SPLINE
SPL {X  -159.990, Y  +513.606, Z    +0.000, E1  +339.879, E3 -411702.660}
SPL {X  -159.990, Y  +508.660, Z    +0.000, E1  +338.515, E3 -411718.090}
SPL {X  -159.990, Y  +505.237, Z    +0.000, E1  +337.606, E3 -411728.347}
SPL {X  -159.990, Y  +501.963, Z    +0.000, E1  +336.712, E3 -411737.451}
SPL {X  -159.990, Y  +498.406, Z    +0.000, E1  +335.789, E3 -411747.202}
SPL {X  -159.990, Y  +494.693, Z    +0.000, E1  +334.929, E3 -411757.669}
SPL {X  -159.990, Y  +491.649, Z    +0.000, E1  +334.596, E3 -411768.871}
SPL {X  -159.990, Y  +488.807, Z    +0.000, E1  +334.603, E3 -411781.596}
SPL {X  -159.990, Y  +486.070, Z    +0.000, E1  +334.601, E3 -411793.827}
SPL {X  -159.990, Y  +483.747, Z    +0.000, E1  +334.616, E3 -411804.240}
SPL {X  -159.990, Y  +481.980, Z    +0.000, E1  +334.616, E3 -411812.137}
SPL {X  -159.990, Y  +479.252, Z    +0.000, E1  +334.588, E3 -411824.279}
SPL {X  -159.990, Y  +475.940, Z    +0.000, E1  +334.597, E3 -411839.099}
SPL {X  -159.990, Y  +473.026, Z    +0.000, E1  +334.601, E3 -411852.129}
SPL {X  -159.990, Y  +470.047, Z    +0.000, E1  +334.598, E3 -411865.447}
SPL {X  -159.990, Y  +466.213, Z    +0.000, E1  +334.567, E3 -411882.527}
SPL {X  -159.990, Y  +462.520, Z    +0.000, E1  +334.600, E3 -411899.096}
SPL {X  -159.990, Y  +460.081, Z    +0.000, E1  +334.610, E3 -411909.997}
SPL {X  -159.990, Y  +457.497, Z    +0.000, E1  +334.597, E3 -411921.522}
SPL {X  -159.990, Y  +455.126, Z    +0.000, E1  +334.611, E3 -411932.130}
SPL {X  -159.990, Y  +452.123, Z    +0.000, E1  +334.574, E3 -411945.488}
SPL {X  -159.990, Y  +448.503, Z    +0.000, E1  +334.590, E3 -411961.689}
SPL {X  -159.990, Y  +445.882, Z    +0.000, E1  +334.615, E3 -411973.492}
SPL {X  -159.990, Y  +443.345, Z    +0.000, E1  +334.610, E3 -411984.874}
SPL {X  -159.990, Y  +441.077, Z    +0.000, E1  +334.631, E3 -411995.072}
SPL {X  -159.990, Y  +438.608, Z    +0.000, E1  +334.608, E3 -412006.069}
SPL {X  -159.990, Y  +435.579, Z    +0.000, E1  +334.614, E3 -412019.623}
SPL {X  -159.990, Y  +432.613, Z    +0.000, E1  +334.610, E3 -412032.890}
SPL {X  -159.990, Y  +429.079, Z    +0.000, E1  +334.593, E3 -412048.661}
SPL {X  -159.990, Y  +426.149, Z    +0.000, E1  +334.626, E3 -412061.823}
SPL {X  -159.990, Y  +423.417, Z    +0.000, E1  +334.600, E3 -412073.989}
SPL {X  -159.990, Y  +419.467, Z    +0.000, E1  +334.583, E3 -412091.623}
SPL {X  -159.990, Y  +416.355, Z    +0.000, E1  +334.625, E3 -412105.621}
SPL {X  -159.990, Y  +413.684, Z    +0.000, E1  +334.603, E3 -412117.527}
SPL {X  -159.990, Y  +410.645, Z    +0.000, E1  +334.615, E3 -412131.139}
SPL {X  -159.990, Y  +408.351, Z    +0.000, E1  +334.628, E3 -412141.425}
SPL {X  -159.990, Y  +406.574, Z    +0.000, E1  +334.625, E3 -412149.342}
SPL {X  -159.990, Y  +404.255, Z    +0.000, E1  +334.609, E3 -412159.678}
SPL {X  -159.990, Y  +401.103, Z    +0.000, E1  +334.596, E3 -412173.742}
SPL {X  -159.990, Y  +398.389, Z    +0.000, E1  +334.619, E3 -412185.938}
SPL {X  -159.990, Y  +395.411, Z    +0.000, E1  +334.600, E3 -412199.235}
SPL {X  -159.990, Y  +392.473, Z    +0.000, E1  +334.623, E3 -412212.421}
SPL {X  -159.990, Y  +390.187, Z    +0.000, E1  +334.622, E3 -412222.679}
SPL {X  -159.990, Y  +387.503, Z    +0.000, E1  +334.622, E3 -412234.673}
SPL {X  -159.990, Y  +384.711, Z    +0.000, E1  +334.612, E3 -412247.117}
SPL {X  -159.988, Y  +381.794, Z    +0.000, E1  +334.611, E3 -412260.152}
SPL {X  -159.958, Y  +379.279, Z    +0.000, E1  +334.625, E3 -412271.442}
SPL {X  -159.867, Y  +376.223, Z    +0.000, E1  +334.608, E3 -412285.157}
SPL {X  -159.727, Y  +373.325, Z    +0.000, E1  +334.659, E3 -412298.322}
SPL {X  -159.549, Y  +370.634, Z    +0.000, E1  +334.653, E3 -412310.495}
SPL {X  -159.201, Y  +366.633, Z    +0.000, E1  +334.686, E3 -412328.687}
SPL {X  -158.798, Y  +363.007, Z    +0.000, E1  +334.761, E3 -412345.345}
SPL {X  -158.453, Y  +360.380, Z    +0.000, E1  +334.828, E3 -412357.489}
SPL {X  -158.127, Y  +358.155, Z    +0.000, E1  +334.874, E3 -412367.820}
SPL {X  -158.095, Y  +357.947, Z    +0.000, E1  +338.259, E3 -412399.392}
ENDSPLINE

SPLINE
SPL {X  -158.454, Y  +360.384, Z    +0.000, E1  +340.634, E3 -412411.543}
SPL {X  -159.737, Y  +373.507, Z    +0.000, E1  +349.689, E3 -412433.579}
SPL {X  -159.990, Y  +382.574, Z    +0.000, E1  +355.537, E3 -412440.266}
SPL {X  -159.990, Y  +387.496, Z    +0.000, E1  +358.996, E3 -412443.012}
SPL {X  -159.990, Y  +395.121, Z    +0.000, E1  +364.514, E3 -412447.324}
SPL {X  -159.990, Y  +407.941, Z    +0.000, E1  +374.126, E3 -412459.398}
SPL {X  -159.990, Y  +418.671, Z    +0.000, E1  +379.855, E3 -412478.814}
SPL {X  -159.990, Y  +429.878, Z    +0.000, E1  +383.330, E3 -412508.869}
SPL {X  -159.990, Y  +432.766, Z    +0.000, E1  +383.321, E3 -412523.092}
SPL {X  -159.990, Y  +434.794, Z    +0.000, E1  +383.304, E3 -412533.123}
SPL {X  -159.990, Y  +437.007, Z    +0.000, E1  +383.323, E3 -412543.976}
SPL {X  -159.990, Y  +439.778, Z    +0.000, E1  +383.323, E3 -412557.608}
SPL {X  -159.990, Y  +442.010, Z    +0.000, E1  +383.308, E3 -412568.629}
SPL {X  -159.990, Y  +443.729, Z    +0.000, E1  +383.310, E3 -412577.085}
SPL {X  -159.990, Y  +446.037, Z    +0.000, E1  +383.324, E3 -412588.422}
SPL {X  -159.990, Y  +448.341, Z    +0.000, E1  +383.317, E3 -412599.740}
SPL {X  -159.990, Y  +450.345, Z    +0.000, E1  +383.316, E3 -412609.618}
SPL {X  -159.990, Y  +452.828, Z    +0.000, E1  +383.330, E3 -412621.817}
SPL {X  -159.990, Y  +456.338, Z    +0.000, E1  +383.359, E3 -412639.009}
SPL {X  -159.990, Y  +459.480, Z    +0.000, E1  +383.323, E3 -412654.551}
SPL {X  -159.990, Y  +461.803, Z    +0.000, E1  +383.322, E3 -412665.986}
SPL {X  -159.990, Y  +464.971, Z    +0.000, E1  +383.357, E3 -412681.492}
SPL {X  -159.990, Y  +467.934, Z    +0.000, E1  +383.321, E3 -412696.149}
SPL {X  -159.990, Y  +469.939, Z    +0.000, E1  +383.319, E3 -412706.011}
SPL {X  -159.990, Y  +472.144, Z    +0.000, E1  +383.327, E3 -412716.862}
SPL {X  -159.990, Y  +474.152, Z    +0.000, E1  +383.309, E3 -412726.814}
SPL {X  -159.990, Y  +476.560, Z    +0.000, E1  +383.332, E3 -412738.622}
SPL {X  -159.990, Y  +478.770, Z    +0.000, E1  +383.306, E3 -412749.547}
SPL {X  -159.990, Y  +480.905, Z    +0.000, E1  +383.327, E3 -412760.015}
SPL {X  -159.990, Y  +484.251, Z    +0.000, E1  +383.352, E3 -412776.430}
SPL {X  -159.990, Y  +488.031, Z    +0.000, E1  +383.345, E3 -412795.063}
SPL {X  -159.990, Y  +491.121, Z    +0.000, E1  +383.323, E3 -412810.309}
SPL {X  -159.990, Y  +493.610, Z    +0.000, E1  +383.323, E3 -412822.562}
SPL {X  -159.990, Y  +496.863, Z    +0.000, E1  +383.350, E3 -412838.522}
SPL {X  -159.990, Y  +499.995, Z    +0.000, E1  +383.324, E3 -412853.983}
SPL {X  -159.990, Y  +502.341, Z    +0.000, E1  +383.320, E3 -412865.542}
SPL {X  -159.990, Y  +504.419, Z    +0.000, E1  +383.313, E3 -412875.784}
SPL {X  -159.990, Y  +507.187, Z    +0.000, E1  +383.346, E3 -412889.337}
SPL {X  -159.990, Y  +510.344, Z    +0.000, E1  +383.327, E3 -412904.922}
SPL {X  -159.990, Y  +512.484, Z    +0.000, E1  +383.309, E3 -412915.494}
SPL {X  -159.990, Y  +514.016, Z    +0.000, E1  +383.308, E3 -412923.043}
SPL {X  -159.990, Y  +516.195, Z    +0.000, E1  +383.325, E3 -412933.731}
SPL {X  -159.990, Y  +518.925, Z    +0.000, E1  +383.333, E3 -412947.094}
SPL {X  -159.990, Y  +521.408, Z    +0.000, E1  +383.329, E3 -412959.303}
SPL {X  -159.990, Y  +523.942, Z    +0.000, E1  +383.333, E3 -412971.796}
SPL {X  -159.990, Y  +527.007, Z    +0.000, E1  +383.339, E3 -412986.895}
SPL {X  -159.990, Y  +529.993, Z    +0.000, E1  +383.329, E3 -413001.598}
SPL {X  -159.990, Y  +532.441, Z    +0.000, E1  +383.322, E3 -413013.649}
SPL {X  -159.990, Y  +534.618, Z    +0.000, E1  +383.322, E3 -413024.382}
SPL {X  -159.990, Y  +537.024, Z    +0.000, E1  +383.321, E3 -413036.244}
SPL {X  -159.990, Y  +539.129, Z    +0.000, E1  +383.310, E3 -413046.627}
SPL {X  -159.990, Y  +541.183, Z    +0.000, E1  +383.319, E3 -413056.724}
SPL {X  -159.990, Y  +543.647, Z    +0.000, E1  +383.325, E3 -413068.827}
SPL {X  -159.990, Y  +546.832, Z    +0.000, E1  +383.349, E3 -413084.450}
SPL {X  -159.990, Y  +549.756, Z    +0.000, E1  +383.320, E3 -413098.891}
SPL {X  -159.990, Y  +551.655, Z    +0.000, E1  +383.320, E3 -413108.241}
SPL {X  -159.990, Y  +553.711, Z    +0.000, E1  +383.317, E3 -413118.363}
SPL {X  -159.990, Y  +556.481, Z    +0.000, E1  +383.354, E3 -413131.925}
SPL {X  -159.990, Y  +559.475, Z    +0.000, E1  +383.321, E3 -413146.730}
SPL {X  -159.990, Y  +561.830, Z    +0.000, E1  +383.325, E3 -413158.315}
SPL {X  -159.990, Y  +564.273, Z    +0.000, E1  +383.325, E3 -413170.339}
SPL {X  -159.990, Y  +566.342, Z    +0.000, E1  +383.314, E3 -413180.544}
SPL {X  -159.990, Y  +568.184, Z    +0.000, E1  +383.317, E3 -413189.605}
SPL {X  -159.990, Y  +570.314, Z    +0.000, E1  +383.326, E3 -413200.067}
SPL {X  -159.990, Y  +573.444, Z    +0.000, E1  +383.356, E3 -413215.406}
SPL {X  -159.990, Y  +577.161, Z    +0.000, E1  +383.346, E3 -413233.731}
SPL {X  -159.990, Y  +580.840, Z    +0.000, E1  +383.355, E3 -413251.780}
SPL {X  -159.990, Y  +583.973, Z    +0.000, E1  +383.332, E3 -413267.241}
SPL {X  -159.990, Y  +586.020, Z    +0.000, E1  +383.323, E3 -413277.325}
SPL {X  -159.990, Y  +587.711, Z    +0.000, E1  +383.318, E3 -413285.665}
SPL {X  -159.990, Y  +589.763, Z    +0.000, E1  +383.328, E3 -413295.741}
SPL {X  -159.990, Y  +591.698, Z    +0.000, E1  +383.324, E3 -413305.226}
SPL {X  -159.990, Y  +593.847, Z    +0.000, E1  +383.340, E3 -413315.757}
SPL {X  -159.990, Y  +597.018, Z    +0.000, E1  +383.367, E3 -413331.288}
SPL {X  -159.990, Y  +599.887, Z    +0.000, E1  +383.341, E3 -413345.393}
SPL {X  -159.990, Y  +601.949, Z    +0.000, E1  +383.344, E3 -413355.519}
SPL {X  -159.990, Y  +605.106, Z    +0.000, E1  +383.383, E3 -413370.965}
SPL {X  -159.990, Y  +608.111, Z    +0.000, E1  +383.342, E3 -413385.816}
SPL {X  -159.990, Y  +610.073, Z    +0.000, E1  +383.343, E3 -413395.474}
SPL {X  -159.990, Y  +612.330, Z    +0.000, E1  +383.340, E3 -413406.602}
SPL {X  -159.990, Y  +615.036, Z    +0.000, E1  +383.353, E3 -413419.889}
SPL {X  -159.990, Y  +618.481, Z    +0.000, E1  +383.366, E3 -413436.827}
SPL {X  -159.990, Y  +621.517, Z    +0.000, E1  +383.337, E3 -413451.810}
SPL {X  -159.990, Y  +623.764, Z    +0.000, E1  +383.335, E3 -413462.861}
SPL {X  -159.990, Y  +626.608, Z    +0.000, E1  +383.361, E3 -413476.786}
SPL {X  -159.990, Y  +630.271, Z    +0.000, E1  +383.375, E3 -413494.747}
SPL {X  -159.990, Y  +633.318, Z    +0.000, E1  +383.339, E3 -413509.824}
SPL {X  -159.990, Y  +635.650, Z    +0.000, E1  +383.339, E3 -413521.295}
SPL {X  -159.990, Y  +638.406, Z    +0.000, E1  +383.354, E3 -413534.862}
SPL {X  -159.990, Y  +641.831, Z    +0.000, E1  +383.342, E3 -413551.809}
SPL {X  -159.990, Y  +644.884, Z    +0.000, E1  +383.324, E3 -413566.896}
SPL {X  -159.990, Y  +647.550, Z    +0.000, E1  +383.318, E3 -413580.063}
SPL {X  -159.990, Y  +650.790, Z    +0.000, E1  +383.346, E3 -413595.930}
SPL {X  -159.990, Y  +654.543, Z    +0.000, E1  +383.348, E3 -413614.382}
SPL {X  -159.990, Y  +658.319, Z    +0.000, E1  +383.349, E3 -413632.972}
SPL {X  -159.990, Y  +661.392, Z    +0.000, E1  +383.318, E3 -413648.175}
SPL {X  -159.990, Y  +663.662, Z    +0.000, E1  +383.322, E3 -413659.299}
SPL {X  -159.990, Y  +665.964, Z    +0.000, E1  +383.328, E3 -413670.590}
SPL {X  -159.990, Y  +667.870, Z    +0.000, E1  +383.320, E3 -413679.996}
SPL {X  -159.990, Y  +669.861, Z    +0.000, E1  +383.321, E3 -413689.798}
SPL {X  -159.983, Y  +672.946, Z    +0.000, E1  +383.359, E3 -413704.907}
SPL {X  -159.924, Y  +676.110, Z    +0.000, E1  +383.320, E3 -413720.606}
SPL {X  -159.845, Y  +678.302, Z    +0.000, E1  +383.298, E3 -413731.508}
SPL {X  -159.760, Y  +680.081, Z    +0.000, E1  +383.288, E3 -413740.352}
SPL {X  -159.626, Y  +682.287, Z    +0.000, E1  +383.280, E3 -413751.323}
SPL {X  -159.462, Y  +684.486, Z    +0.000, E1  +383.258, E3 -413762.323}
SPL {X  -159.212, Y  +687.262, Z    +0.000, E1  +383.238, E3 -413776.227}
SPL {X  -158.971, Y  +689.529, Z    +0.000, E1  +383.181, E3 -413787.686}
SPL {X  -158.658, Y  +692.098, Z    +0.000, E1  +383.176, E3 -413800.593}
ENDSPLINE

SPLINE
SPL {X  -159.063, Y  +688.696, Z    +0.000, E1  +377.094, E3 -413842.811}
SPL {X  -159.987, Y  +672.488, Z    +0.000, E1  +365.638, E3 -413866.876}
SPL {X  -159.990, Y  +663.928, Z    +0.000, E1  +359.662, E3 -413872.671}
SPL {X  -159.990, Y  +658.009, Z    +0.000, E1  +355.226, E3 -413876.371}
SPL {X  -159.990, Y  +651.879, Z    +0.000, E1  +350.548, E3 -413881.433}
SPL {X  -159.990, Y  +637.832, Z    +0.000, E1  +341.694, E3 -413899.024}
SPL {X  -159.990, Y  +626.634, Z    +0.000, E1  +337.968, E3 -413929.877}
SPL {X  -159.990, Y  +624.622, Z    +0.000, E1  +337.980, E3 -413940.461}
SPL {X  -159.990, Y  +622.489, Z    +0.000, E1  +337.969, E3 -413951.628}
SPL {X  -159.990, Y  +619.955, Z    +0.000, E1  +337.968, E3 -413964.918}
SPL {X  -159.990, Y  +617.386, Z    +0.000, E1  +337.968, E3 -413978.392}
SPL {X  -159.990, Y  +614.863, Z    +0.000, E1  +337.969, E3 -413991.625}
SPL {X  -159.990, Y  +612.600, Z    +0.000, E1  +337.975, E3 -414003.509}
SPL {X  -159.990, Y  +610.646, Z    +0.000, E1  +337.979, E3 -414013.766}
SPL {X  -159.990, Y  +608.810, Z    +0.000, E1  +337.977, E3 -414023.399}
SPL {X  -159.990, Y  +605.804, Z    +0.000, E1  +337.936, E3 -414039.044}
SPL {X  -159.990, Y  +602.819, Z    +0.000, E1  +337.963, E3 -414054.715}
SPL {X  -159.990, Y  +600.642, Z    +0.000, E1  +337.968, E3 -414066.143}
SPL {X  -159.990, Y  +598.568, Z    +0.000, E1  +337.954, E3 -414076.936}
SPL {X  -159.990, Y  +596.440, Z    +0.000, E1  +337.964, E3 -414088.118}
SPL {X  -159.990, Y  +593.768, Z    +0.000, E1  +337.929, E3 -414102.051}
SPL {X  -159.990, Y  +590.068, Z    +0.000, E1  +337.924, E3 -414121.419}
SPL {X  -159.990, Y  +586.620, Z    +0.000, E1  +337.935, E3 -414139.482}
SPL {X  -159.990, Y  +584.080, Z    +0.000, E1  +337.953, E3 -414152.808}
SPL {X  -159.990, Y  +581.924, Z    +0.000, E1  +337.949, E3 -414164.108}
SPL {X  -159.990, Y  +578.886, Z    +0.000, E1  +337.918, E3 -414179.962}
SPL {X  -159.990, Y  +576.252, Z    +0.000, E1  +337.962, E3 -414193.860}
SPL {X  -159.990, Y  +574.188, Z    +0.000, E1  +337.947, E3 -414204.633}
SPL {X  -159.990, Y  +571.954, Z    +0.000, E1  +337.959, E3 -414216.391}
SPL {X  -159.990, Y  +570.110, Z    +0.000, E1  +337.958, E3 -414226.041}
SPL {X  -159.990, Y  +568.165, Z    +0.000, E1  +337.957, E3 -414236.221}
SPL {X  -159.990, Y  +566.106, Z    +0.000, E1  +337.954, E3 -414247.004}
SPL {X  -159.990, Y  +563.259, Z    +0.000, E1  +337.929, E3 -414261.886}
SPL {X  -159.990, Y  +559.661, Z    +0.000, E1  +337.922, E3 -414280.709}
SPL {X  -159.990, Y  +555.965, Z    +0.000, E1  +337.915, E3 -414300.018}
SPL {X  -159.990, Y  +553.115, Z    +0.000, E1  +337.946, E3 -414315.003}
SPL {X  -159.990, Y  +550.886, Z    +0.000, E1  +337.944, E3 -414326.685}
SPL {X  -159.990, Y  +548.568, Z    +0.000, E1  +337.944, E3 -414338.806}
SPL {X  -159.990, Y  +545.859, Z    +0.000, E1  +337.926, E3 -414352.955}
SPL {X  -159.990, Y  +543.060, Z    +0.000, E1  +337.943, E3 -414367.679}
SPL {X  -159.990, Y  +539.928, Z    +0.000, E1  +337.917, E3 -414384.020}
SPL {X  -159.990, Y  +536.935, Z    +0.000, E1  +337.942, E3 -414399.737}
SPL {X  -159.990, Y  +534.656, Z    +0.000, E1  +337.946, E3 -414411.681}
SPL {X  -159.990, Y  +531.679, Z    +0.000, E1  +337.913, E3 -414427.195}
SPL {X  -159.990, Y  +527.941, Z    +0.000, E1  +337.907, E3 -414446.737}
SPL {X  -159.990, Y  +525.053, Z    +0.000, E1  +337.942, E3 -414461.927}
SPL {X  -159.990, Y  +522.838, Z    +0.000, E1  +337.933, E3 -414473.531}
SPL {X  -159.990, Y  +519.698, Z    +0.000, E1  +337.916, E3 -414489.915}
SPL {X  -159.990, Y  +517.251, Z    +0.000, E1  +337.946, E3 -414502.774}
SPL {X  -159.990, Y  +515.568, Z    +0.000, E1  +338.084, E3 -414512.871}
ENDSPLINE

SPLINE
SPL {X  -159.990, Y  +517.293, Z    +0.000, E1  +340.923, E3 -414529.170}
ENDSPLINE

SPLINE
SPL {X  -159.990, Y  +512.548, Z    +0.000, E1  +339.587, E3 -414544.745}
SPL {X  -159.990, Y  +508.660, Z    +0.000, E1  +338.515, E3 -414556.799}
SPL {X  -159.990, Y  +503.499, Z    +0.000, E1  +337.116, E3 -414571.878}
SPL {X  -159.990, Y  +498.406, Z    +0.000, E1  +335.789, E3 -414585.911}
SPL {X  -159.990, Y  +494.693, Z    +0.000, E1  +334.929, E3 -414596.379}
SPL {X  -159.990, Y  +491.649, Z    +0.000, E1  +334.596, E3 -414607.581}
SPL {X  -159.990, Y  +488.807, Z    +0.000, E1  +334.603, E3 -414620.306}
SPL {X  -159.990, Y  +486.070, Z    +0.000, E1  +334.601, E3 -414632.537}
SPL {X  -159.990, Y  +482.821, Z    +0.000, E1  +334.589, E3 -414647.038}
SPL {X  -159.990, Y  +480.183, Z    +0.000, E1  +334.616, E3 -414658.878}
SPL {X  -159.990, Y  +478.407, Z    +0.000, E1  +334.616, E3 -414666.819}
SPL {X  -159.990, Y  +475.940, Z    +0.000, E1  +334.597, E3 -414677.809}
SPL {X  -159.990, Y  +473.026, Z    +0.000, E1  +334.601, E3 -414690.839}
SPL {X  -159.990, Y  +470.047, Z    +0.000, E1  +334.598, E3 -414704.157}
SPL {X  -159.990, Y  +467.082, Z    +0.000, E1  +334.601, E3 -414717.404}
SPL {X  -159.990, Y  +464.919, Z    +0.000, E1  +334.619, E3 -414727.131}
SPL {X  -159.990, Y  +462.520, Z    +0.000, E1  +334.600, E3 -414737.805}
SPL {X  -159.990, Y  +460.081, Z    +0.000, E1  +334.610, E3 -414748.707}
SPL {X  -159.990, Y  +457.497, Z    +0.000, E1  +334.597, E3 -414760.231}
SPL {X  -159.990, Y  +454.323, Z    +0.000, E1  +334.588, E3 -414774.390}
SPL {X  -159.990, Y  +451.400, Z    +0.000, E1  +334.603, E3 -414787.481}
SPL {X  -159.990, Y  +448.503, Z    +0.000, E1  +334.590, E3 -414800.399}
SPL {X  -159.990, Y  +445.108, Z    +0.000, E1  +334.593, E3 -414815.637}
SPL {X  -159.990, Y  +441.797, Z    +0.000, E1  +334.610, E3 -414830.516}
SPL {X  -159.990, Y  +439.442, Z    +0.000, E1  +334.631, E3 -414841.093}
SPL {X  -159.990, Y  +436.316, Z    +0.000, E1  +334.580, E3 -414854.975}
SPL {X  -159.990, Y  +432.613, Z    +0.000, E1  +334.610, E3 -414871.600}
SPL {X  -159.990, Y  +429.079, Z    +0.000, E1  +334.593, E3 -414887.371}
SPL {X  -159.990, Y  +426.149, Z    +0.000, E1  +334.626, E3 -414900.533}
SPL {X  -159.990, Y  +423.417, Z    +0.000, E1  +334.600, E3 -414912.698}
SPL {X  -159.990, Y  +419.467, Z    +0.000, E1  +334.583, E3 -414930.333}
SPL {X  -159.990, Y  +416.355, Z    +0.000, E1  +334.625, E3 -414944.330}
SPL {X  -159.990, Y  +413.684, Z    +0.000, E1  +334.603, E3 -414956.237}
SPL {X  -159.990, Y  +410.645, Z    +0.000, E1  +334.615, E3 -414969.849}
SPL {X  -159.990, Y  +408.351, Z    +0.000, E1  +334.628, E3 -414980.135}
SPL {X  -159.990, Y  +406.574, Z    +0.000, E1  +334.625, E3 -414988.052}
SPL {X  -159.990, Y  +404.255, Z    +0.000, E1  +334.609, E3 -414998.388}
SPL {X  -159.990, Y  +401.103, Z    +0.000, E1  +334.596, E3 -415012.452}
SPL {X  -159.990, Y  +398.389, Z    +0.000, E1  +334.619, E3 -415024.648}
SPL {X  -159.990, Y  +395.411, Z    +0.000, E1  +334.600, E3 -415037.945}
SPL {X  -159.990, Y  +392.473, Z    +0.000, E1  +334.623, E3 -415051.130}
SPL {X  -159.990, Y  +390.187, Z    +0.000, E1  +334.622, E3 -415061.388}
SPL {X  -159.990, Y  +387.503, Z    +0.000, E1  +334.622, E3 -415073.383}
SPL {X  -159.990, Y  +384.711, Z    +0.000, E1  +334.612, E3 -415085.827}
SPL {X  -159.988, Y  +381.794, Z    +0.000, E1  +334.611, E3 -415098.862}
SPL {X  -159.958, Y  +379.279, Z    +0.000, E1  +334.625, E3 -415110.152}
SPL {X  -159.894, Y  +376.959, Z    +0.000, E1  +334.630, E3 -415120.596}
SPL {X  -159.765, Y  +374.027, Z    +0.000, E1  +334.633, E3 -415133.812}
SPL {X  -159.607, Y  +371.442, Z    +0.000, E1  +334.673, E3 -415145.587}
SPL {X  -159.379, Y  +368.534, Z    +0.000, E1  +334.684, E3 -415158.774}
SPL {X  -159.113, Y  +365.767, Z    +0.000, E1  +334.734, E3 -415171.414}
SPL {X  -158.869, Y  +363.595, Z    +0.000, E1  +334.770, E3 -415181.385}
SPL {X  -158.527, Y  +360.915, Z    +0.000, E1  +334.798, E3 -415193.692}
SPL {X  -158.127, Y  +358.155, Z    +0.000, E1  +334.874, E3 -415206.530}
SPL {X  -158.095, Y  +357.947, Z    +0.000, E1  +338.259, E3 -415238.102}
ENDSPLINE

SPLINE
SPL {X  -158.454, Y  +360.384, Z    +0.000, E1  +340.634, E3 -415250.253}
SPL {X  -159.737, Y  +373.507, Z    +0.000, E1  +349.689, E3 -415272.288}
SPL {X  -159.990, Y  +382.574, Z    +0.000, E1  +355.537, E3 -415278.976}
SPL {X  -159.990, Y  +387.496, Z    +0.000, E1  +358.996, E3 -415281.721}
SPL {X  -159.990, Y  +395.121, Z    +0.000, E1  +364.514, E3 -415286.033}
SPL {X  -159.990, Y  +407.941, Z    +0.000, E1  +374.126, E3 -415298.108}
SPL {X  -159.990, Y  +418.671, Z    +0.000, E1  +379.855, E3 -415317.524}
SPL {X  -159.990, Y  +429.878, Z    +0.000, E1  +383.330, E3 -415347.579}
SPL {X  -159.990, Y  +432.103, Z    +0.000, E1  +383.301, E3 -415358.598}
SPL {X  -159.990, Y  +434.188, Z    +0.000, E1  +383.325, E3 -415368.794}
SPL {X  -159.990, Y  +436.320, Z    +0.000, E1  +383.304, E3 -415379.347}
SPL {X  -159.990, Y  +439.169, Z    +0.000, E1  +383.353, E3 -415393.264}
SPL {X  -159.990, Y  +442.945, Z    +0.000, E1  +383.339, E3 -415411.882}
SPL {X  -159.990, Y  +446.037, Z    +0.000, E1  +383.324, E3 -415427.132}
SPL {X  -159.990, Y  +448.341, Z    +0.000, E1  +383.317, E3 -415438.449}
SPL {X  -159.990, Y  +450.345, Z    +0.000, E1  +383.316, E3 -415448.327}
SPL {X  -159.990, Y  +452.828, Z    +0.000, E1  +383.330, E3 -415460.527}
SPL {X  -159.990, Y  +456.338, Z    +0.000, E1  +383.359, E3 -415477.719}
SPL {X  -159.990, Y  +459.480, Z    +0.000, E1  +383.323, E3 -415493.260}
SPL {X  -159.990, Y  +461.803, Z    +0.000, E1  +383.322, E3 -415504.695}
SPL {X  -159.990, Y  +464.971, Z    +0.000, E1  +383.357, E3 -415520.201}
SPL {X  -159.990, Y  +467.934, Z    +0.000, E1  +383.321, E3 -415534.859}
SPL {X  -159.990, Y  +469.939, Z    +0.000, E1  +383.319, E3 -415544.720}
SPL {X  -159.990, Y  +472.144, Z    +0.000, E1  +383.327, E3 -415555.571}
SPL {X  -159.990, Y  +474.152, Z    +0.000, E1  +383.309, E3 -415565.523}
SPL {X  -159.990, Y  +475.762, Z    +0.000, E1  +383.308, E3 -415573.453}
SPL {X  -159.990, Y  +478.041, Z    +0.000, E1  +383.328, E3 -415584.628}
SPL {X  -159.990, Y  +480.905, Z    +0.000, E1  +383.327, E3 -415598.724}
SPL {X  -159.990, Y  +483.391, Z    +0.000, E1  +383.320, E3 -415610.965}
SPL {X  -159.990, Y  +485.299, Z    +0.000, E1  +383.310, E3 -415620.394}
SPL {X  -159.990, Y  +487.362, Z    +0.000, E1  +383.320, E3 -415630.528}
SPL {X  -159.990, Y  +490.503, Z    +0.000, E1  +383.351, E3 -415645.923}
SPL {X  -159.990, Y  +493.610, Z    +0.000, E1  +383.323, E3 -415661.272}
SPL {X  -159.990, Y  +495.794, Z    +0.000, E1  +383.312, E3 -415672.045}
SPL {X  -159.990, Y  +497.668, Z    +0.000, E1  +383.317, E3 -415681.255}
SPL {X  -159.990, Y  +499.995, Z    +0.000, E1  +383.324, E3 -415692.693}
SPL {X  -159.990, Y  +502.341, Z    +0.000, E1  +383.320, E3 -415704.252}
SPL {X  -159.990, Y  +504.419, Z    +0.000, E1  +383.313, E3 -415714.493}
SPL {X  -159.990, Y  +506.252, Z    +0.000, E1  +383.313, E3 -415723.519}
SPL {X  -159.990, Y  +508.697, Z    +0.000, E1  +383.335, E3 -415735.502}
SPL {X  -159.990, Y  +511.771, Z    +0.000, E1  +383.331, E3 -415750.649}
SPL {X  -159.990, Y  +514.016, Z    +0.000, E1  +383.308, E3 -415761.753}
SPL {X  -159.990, Y  +516.195, Z    +0.000, E1  +383.325, E3 -415772.440}
SPL {X  -159.990, Y  +518.925, Z    +0.000, E1  +383.333, E3 -415785.804}
SPL {X  -159.990, Y  +521.408, Z    +0.000, E1  +383.329, E3 -415798.013}
SPL {X  -159.990, Y  +523.942, Z    +0.000, E1  +383.333, E3 -415810.506}
SPL {X  -159.990, Y  +526.221, Z    +0.000, E1  +383.314, E3 -415821.782}
SPL {X  -159.990, Y  +527.834, Z    +0.000, E1  +383.311, E3 -415829.732}
SPL {X  -159.990, Y  +529.993, Z    +0.000, E1  +383.329, E3 -415840.308}
SPL {X  -159.990, Y  +532.441, Z    +0.000, E1  +383.322, E3 -415852.358}
SPL {X  -159.990, Y  +534.618, Z    +0.000, E1  +383.322, E3 -415863.091}
SPL {X  -159.990, Y  +537.024, Z    +0.000, E1  +383.321, E3 -415874.954}
SPL {X  -159.990, Y  +539.129, Z    +0.000, E1  +383.310, E3 -415885.337}
SPL {X  -159.990, Y  +541.183, Z    +0.000, E1  +383.319, E3 -415895.433}
SPL {X  -159.990, Y  +543.647, Z    +0.000, E1  +383.325, E3 -415907.536}
SPL {X  -159.990, Y  +546.832, Z    +0.000, E1  +383.349, E3 -415923.159}
SPL {X  -159.990, Y  +549.756, Z    +0.000, E1  +383.320, E3 -415937.600}
SPL {X  -159.990, Y  +551.655, Z    +0.000, E1  +383.320, E3 -415946.951}
SPL {X  -159.990, Y  +553.711, Z    +0.000, E1  +383.317, E3 -415957.073}
SPL {X  -159.990, Y  +555.637, Z    +0.000, E1  +383.323, E3 -415966.542}
SPL {X  -159.990, Y  +558.758, Z    +0.000, E1  +383.351, E3 -415981.851}
SPL {X  -159.990, Y  +561.830, Z    +0.000, E1  +383.325, E3 -415997.025}
SPL {X  -159.990, Y  +564.273, Z    +0.000, E1  +383.325, E3 -416009.049}
SPL {X  -159.990, Y  +567.351, Z    +0.000, E1  +383.348, E3 -416024.145}
SPL {X  -159.990, Y  +570.314, Z    +0.000, E1  +383.326, E3 -416038.777}
SPL {X  -159.990, Y  +572.504, Z    +0.000, E1  +383.321, E3 -416049.562}
SPL {X  -159.990, Y  +575.653, Z    +0.000, E1  +383.355, E3 -416064.999}
SPL {X  -159.990, Y  +578.932, Z    +0.000, E1  +383.330, E3 -416081.181}
SPL {X  -159.990, Y  +581.497, Z    +0.000, E1  +383.329, E3 -416093.766}
SPL {X  -159.990, Y  +583.973, Z    +0.000, E1  +383.332, E3 -416105.951}
SPL {X  -159.990, Y  +586.020, Z    +0.000, E1  +383.323, E3 -416116.035}
SPL {X  -159.990, Y  +587.711, Z    +0.000, E1  +383.318, E3 -416124.375}
SPL {X  -159.990, Y  +589.763, Z    +0.000, E1  +383.328, E3 -416134.451}
SPL {X  -159.990, Y  +591.698, Z    +0.000, E1  +383.324, E3 -416143.936}
SPL {X  -159.990, Y  +593.847, Z    +0.000, E1  +383.340, E3 -416154.466}
SPL {X  -159.990, Y  +597.018, Z    +0.000, E1  +383.367, E3 -416169.998}
SPL {X  -159.990, Y  +599.887, Z    +0.000, E1  +383.341, E3 -416184.102}
SPL {X  -159.990, Y  +601.949, Z    +0.000, E1  +383.344, E3 -416194.229}
SPL {X  -159.990, Y  +605.106, Z    +0.000, E1  +383.383, E3 -416209.675}
SPL {X  -159.990, Y  +608.111, Z    +0.000, E1  +383.342, E3 -416224.526}
SPL {X  -159.990, Y  +610.073, Z    +0.000, E1  +383.343, E3 -416234.184}
SPL {X  -159.990, Y  +612.330, Z    +0.000, E1  +383.340, E3 -416245.312}
SPL {X  -159.990, Y  +615.036, Z    +0.000, E1  +383.353, E3 -416258.599}
SPL {X  -159.990, Y  +618.481, Z    +0.000, E1  +383.366, E3 -416275.537}
SPL {X  -159.990, Y  +621.517, Z    +0.000, E1  +383.337, E3 -416290.520}
SPL {X  -159.990, Y  +623.764, Z    +0.000, E1  +383.335, E3 -416301.570}
SPL {X  -159.990, Y  +626.608, Z    +0.000, E1  +383.361, E3 -416315.495}
SPL {X  -159.990, Y  +630.271, Z    +0.000, E1  +383.375, E3 -416333.456}
SPL {X  -159.990, Y  +633.318, Z    +0.000, E1  +383.339, E3 -416348.534}
SPL {X  -159.990, Y  +635.650, Z    +0.000, E1  +383.339, E3 -416360.005}
SPL {X  -159.990, Y  +638.406, Z    +0.000, E1  +383.354, E3 -416373.571}
SPL {X  -159.990, Y  +641.131, Z    +0.000, E1  +383.320, E3 -416387.096}
SPL {X  -159.990, Y  +644.241, Z    +0.000, E1  +383.355, E3 -416402.374}
SPL {X  -159.990, Y  +648.287, Z    +0.000, E1  +383.349, E3 -416422.331}
SPL {X  -159.990, Y  +651.427, Z    +0.000, E1  +383.319, E3 -416437.826}
SPL {X  -159.990, Y  +653.536, Z    +0.000, E1  +383.313, E3 -416448.207}
SPL {X  -159.990, Y  +656.380, Z    +0.000, E1  +383.347, E3 -416462.143}
SPL {X  -159.990, Y  +659.180, Z    +0.000, E1  +383.314, E3 -416475.991}
SPL {X  -159.990, Y  +661.392, Z    +0.000, E1  +383.318, E3 -416486.885}
SPL {X  -159.990, Y  +663.662, Z    +0.000, E1  +383.322, E3 -416498.009}
SPL {X  -159.990, Y  +665.964, Z    +0.000, E1  +383.328, E3 -416509.299}
SPL {X  -159.990, Y  +668.989, Z    +0.000, E1  +383.359, E3 -416524.135}
SPL {X  -159.983, Y  +672.946, Z    +0.000, E1  +383.359, E3 -416543.616}
SPL {X  -159.924, Y  +676.110, Z    +0.000, E1  +383.320, E3 -416559.316}
SPL {X  -159.845, Y  +678.302, Z    +0.000, E1  +383.298, E3 -416570.218}
SPL {X  -159.760, Y  +680.081, Z    +0.000, E1  +383.288, E3 -416579.061}
SPL {X  -159.626, Y  +682.287, Z    +0.000, E1  +383.280, E3 -416590.033}
SPL {X  -159.462, Y  +684.486, Z    +0.000, E1  +383.258, E3 -416601.032}
SPL {X  -159.289, Y  +686.457, Z    +0.000, E1  +383.223, E3 -416610.943}
SPL {X  -159.052, Y  +688.801, Z    +0.000, E1  +383.217, E3 -416622.677}
SPL {X  -158.770, Y  +691.222, Z    +0.000, E1  +383.158, E3 -416634.935}
SPL {X  -158.553, Y  +692.896, Z    +0.000, E1  +383.130, E3 -416643.400}
ENDSPLINE

SPLINE
SPL {X  -158.898, Y  +690.164, Z    +0.000, E1  +378.236, E3 -416676.756}
SPL {X  -159.149, Y  +687.882, Z    +0.000, E1  +376.368, E3 -416684.044}
SPL {X  -159.987, Y  +672.488, Z    +0.000, E1  +365.638, E3 -416705.586}
SPL {X  -159.990, Y  +663.928, Z    +0.000, E1  +359.662, E3 -416711.381}
SPL {X  -159.990, Y  +658.009, Z    +0.000, E1  +355.226, E3 -416715.080}
SPL {X  -159.990, Y  +651.879, Z    +0.000, E1  +350.548, E3 -416720.143}
SPL {X  -159.990, Y  +637.832, Z    +0.000, E1  +341.694, E3 -416737.734}
SPL {X  -159.990, Y  +626.634, Z    +0.000, E1  +337.968, E3 -416768.587}
SPL {X  -159.990, Y  +624.622, Z    +0.000, E1  +337.980, E3 -416779.171}
SPL {X  -159.990, Y  +622.489, Z    +0.000, E1  +337.969, E3 -416790.337}
SPL {X  -159.990, Y  +619.955, Z    +0.000, E1  +337.968, E3 -416803.627}
SPL {X  -159.990, Y  +617.386, Z    +0.000, E1  +337.968, E3 -416817.102}
SPL {X  -159.990, Y  +614.863, Z    +0.000, E1  +337.969, E3 -416830.334}
SPL {X  -159.990, Y  +612.600, Z    +0.000, E1  +337.975, E3 -416842.218}
SPL {X  -159.990, Y  +610.646, Z    +0.000, E1  +337.979, E3 -416852.476}
SPL {X  -159.990, Y  +608.810, Z    +0.000, E1  +337.977, E3 -416862.109}
SPL {X  -159.990, Y  +605.804, Z    +0.000, E1  +337.936, E3 -416877.754}
SPL {X  -159.990, Y  +602.819, Z    +0.000, E1  +337.963, E3 -416893.425}
SPL {X  -159.990, Y  +600.642, Z    +0.000, E1  +337.968, E3 -416904.853}
SPL {X  -159.990, Y  +598.568, Z    +0.000, E1  +337.954, E3 -416915.646}
SPL {X  -159.990, Y  +596.440, Z    +0.000, E1  +337.964, E3 -416926.827}
SPL {X  -159.990, Y  +593.768, Z    +0.000, E1  +337.929, E3 -416940.760}
SPL {X  -159.990, Y  +590.068, Z    +0.000, E1  +337.924, E3 -416960.129}
SPL {X  -159.990, Y  +586.620, Z    +0.000, E1  +337.935, E3 -416978.191}
SPL {X  -159.990, Y  +584.080, Z    +0.000, E1  +337.953, E3 -416991.518}
SPL {X  -159.990, Y  +581.924, Z    +0.000, E1  +337.949, E3 -417002.818}
SPL {X  -159.990, Y  +578.886, Z    +0.000, E1  +337.918, E3 -417018.672}
SPL {X  -159.990, Y  +576.252, Z    +0.000, E1  +337.962, E3 -417032.570}
SPL {X  -159.990, Y  +574.188, Z    +0.000, E1  +337.947, E3 -417043.343}
SPL {X  -159.990, Y  +571.954, Z    +0.000, E1  +337.959, E3 -417055.100}
SPL {X  -159.990, Y  +570.110, Z    +0.000, E1  +337.958, E3 -417064.751}
SPL {X  -159.990, Y  +568.165, Z    +0.000, E1  +337.957, E3 -417074.931}
SPL {X  -159.990, Y  +565.292, Z    +0.000, E1  +337.922, E3 -417089.908}
SPL {X  -159.990, Y  +562.598, Z    +0.000, E1  +337.958, E3 -417104.120}
SPL {X  -159.990, Y  +560.652, Z    +0.000, E1  +337.962, E3 -417114.332}
SPL {X  -159.990, Y  +558.143, Z    +0.000, E1  +337.928, E3 -417127.364}
SPL {X  -159.990, Y  +555.329, Z    +0.000, E1  +337.943, E3 -417142.108}
SPL {X  -159.990, Y  +553.115, Z    +0.000, E1  +337.946, E3 -417153.713}
SPL {X  -159.990, Y  +550.886, Z    +0.000, E1  +337.944, E3 -417165.394}
SPL {X  -159.990, Y  +548.568, Z    +0.000, E1  +337.944, E3 -417177.516}
SPL {X  -159.990, Y  +545.859, Z    +0.000, E1  +337.926, E3 -417191.665}
SPL {X  -159.990, Y  +543.060, Z    +0.000, E1  +337.943, E3 -417206.389}
SPL {X  -159.990, Y  +539.928, Z    +0.000, E1  +337.917, E3 -417222.730}
SPL {X  -159.990, Y  +536.935, Z    +0.000, E1  +337.942, E3 -417238.447}
SPL {X  -159.990, Y  +534.656, Z    +0.000, E1  +337.946, E3 -417250.390}
SPL {X  -159.990, Y  +531.679, Z    +0.000, E1  +337.913, E3 -417265.904}
SPL {X  -159.990, Y  +527.941, Z    +0.000, E1  +337.907, E3 -417285.447}
SPL {X  -159.990, Y  +525.053, Z    +0.000, E1  +337.942, E3 -417300.637}
SPL {X  -159.990, Y  +522.838, Z    +0.000, E1  +337.933, E3 -417312.241}
SPL {X  -159.990, Y  +519.698, Z    +0.000, E1  +337.916, E3 -417328.624}
SPL {X  -159.990, Y  +517.251, Z    +0.000, E1  +337.946, E3 -417341.484}
SPL {X  -159.990, Y  +515.568, Z    +0.000, E1  +338.084, E3 -417351.581}
ENDSPLINE

SPLINE
SPL {X  -159.990, Y  +517.293, Z    +0.000, E1  +340.923, E3 -417367.879}
ENDSPLINE

SPLINE
SPL {X  -159.990, Y  +512.548, Z    +0.000, E1  +339.587, E3 -417383.454}
SPL {X  -159.990, Y  +508.660, Z    +0.000, E1  +338.515, E3 -417395.509}
SPL {X  -159.990, Y  +503.499, Z    +0.000, E1  +337.116, E3 -417410.588}
SPL {X  -159.990, Y  +498.406, Z    +0.000, E1  +335.789, E3 -417424.621}
SPL {X  -159.990, Y  +494.693, Z    +0.000, E1  +334.929, E3 -417435.088}
SPL {X  -159.990, Y  +491.649, Z    +0.000, E1  +334.596, E3 -417446.291}
SPL {X  -159.990, Y  +488.807, Z    +0.000, E1  +334.603, E3 -417459.015}
SPL {X  -159.990, Y  +486.070, Z    +0.000, E1  +334.601, E3 -417471.246}
SPL {X  -159.990, Y  +482.821, Z    +0.000, E1  +334.589, E3 -417485.748}
SPL {X  -159.990, Y  +480.183, Z    +0.000, E1  +334.616, E3 -417497.588}
SPL {X  -159.990, Y  +478.407, Z    +0.000, E1  +334.616, E3 -417505.528}
SPL {X  -159.990, Y  +475.940, Z    +0.000, E1  +334.597, E3 -417516.519}
SPL {X  -159.990, Y  +473.026, Z    +0.000, E1  +334.601, E3 -417529.548}
SPL {X  -159.990, Y  +470.047, Z    +0.000, E1  +334.598, E3 -417542.867}
SPL {X  -159.990, Y  +466.213, Z    +0.000, E1  +334.567, E3 -417559.946}
SPL {X  -159.990, Y  +462.520, Z    +0.000, E1  +334.600, E3 -417576.515}
SPL {X  -159.990, Y  +460.081, Z    +0.000, E1  +334.610, E3 -417587.416}
SPL {X  -159.990, Y  +457.497, Z    +0.000, E1  +334.597, E3 -417598.941}
SPL {X  -159.990, Y  +455.126, Z    +0.000, E1  +334.611, E3 -417609.549}
SPL {X  -159.990, Y  +453.438, Z    +0.000, E1  +334.615, E3 -417617.109}
SPL {X  -159.990, Y  +450.823, Z    +0.000, E1  +334.583, E3 -417628.729}
SPL {X  -159.990, Y  +446.894, Z    +0.000, E1  +334.572, E3 -417646.286}
SPL {X  -159.990, Y  +443.345, Z    +0.000, E1  +334.610, E3 -417662.293}
SPL {X  -159.990, Y  +441.077, Z    +0.000, E1  +334.631, E3 -417672.492}
SPL {X  -159.990, Y  +438.608, Z    +0.000, E1  +334.608, E3 -417683.488}
SPL {X  -159.990, Y  +434.852, Z    +0.000, E1  +334.585, E3 -417700.243}
SPL {X  -159.990, Y  +431.966, Z    +0.000, E1  +334.629, E3 -417713.241}
SPL {X  -159.990, Y  +429.079, Z    +0.000, E1  +334.593, E3 -417726.080}
SPL {X  -159.990, Y  +426.149, Z    +0.000, E1  +334.626, E3 -417739.243}
SPL {X  -159.990, Y  +423.417, Z    +0.000, E1  +334.600, E3 -417751.408}
SPL {X  -159.990, Y  +419.467, Z    +0.000, E1  +334.583, E3 -417769.043}
SPL {X  -159.990, Y  +415.368, Z    +0.000, E1  +334.593, E3 -417787.397}
SPL {X  -159.990, Y  +411.297, Z    +0.000, E1  +334.587, E3 -417805.592}
SPL {X  -159.990, Y  +407.450, Z    +0.000, E1  +334.599, E3 -417822.807}
SPL {X  -159.990, Y  +404.255, Z    +0.000, E1  +334.609, E3 -417837.098}
SPL {X  -159.990, Y  +401.103, Z    +0.000, E1  +334.596, E3 -417851.162}
SPL {X  -159.990, Y  +397.743, Z    +0.000, E1  +334.600, E3 -417866.212}
SPL {X  -159.990, Y  +394.848, Z    +0.000, E1  +334.621, E3 -417879.213}
SPL {X  -159.990, Y  +392.473, Z    +0.000, E1  +334.623, E3 -417889.840}
SPL {X  -159.990, Y  +390.187, Z    +0.000, E1  +334.622, E3 -417900.098}
SPL {X  -159.990, Y  +387.503, Z    +0.000, E1  +334.622, E3 -417912.093}
SPL {X  -159.990, Y  +384.711, Z    +0.000, E1  +334.612, E3 -417924.537}
SPL {X  -159.988, Y  +381.794, Z    +0.000, E1  +334.611, E3 -417937.571}
SPL {X  -159.958, Y  +379.279, Z    +0.000, E1  +334.625, E3 -417948.862}
SPL {X  -159.867, Y  +376.223, Z    +0.000, E1  +334.608, E3 -417962.576}
SPL {X  -159.727, Y  +373.325, Z    +0.000, E1  +334.659, E3 -417975.741}
SPL {X  -159.549, Y  +370.634, Z    +0.000, E1  +334.653, E3 -417987.914}
SPL {X  -159.201, Y  +366.633, Z    +0.000, E1  +334.686, E3 -418006.106}
SPL {X  -158.869, Y  +363.595, Z    +0.000, E1  +334.770, E3 -418020.095}
SPL {X  -158.527, Y  +360.915, Z    +0.000, E1  +334.798, E3 -418032.401}
SPL {X  -158.127, Y  +358.155, Z    +0.000, E1  +334.874, E3 -418045.239}
SPL {X  -158.095, Y  +357.947, Z    +0.000, E1  +338.259, E3 -418076.812}
ENDSPLINE

SPLINE
SPL {X  -158.454, Y  +360.384, Z    +0.000, E1  +340.634, E3 -418088.963}
SPL {X  -159.737, Y  +373.507, Z    +0.000, E1  +349.689, E3 -418110.998}
SPL {X  -159.990, Y  +382.574, Z    +0.000, E1  +355.537, E3 -418117.686}
SPL {X  -159.990, Y  +387.496, Z    +0.000, E1  +358.996, E3 -418120.431}
SPL {X  -159.990, Y  +395.121, Z    +0.000, E1  +364.514, E3 -418124.743}
SPL {X  -159.990, Y  +407.941, Z    +0.000, E1  +374.126, E3 -418136.817}
SPL {X  -159.990, Y  +418.671, Z    +0.000, E1  +379.855, E3 -418156.234}
SPL {X  -159.990, Y  +429.878, Z    +0.000, E1  +383.330, E3 -418186.289}
SPL {X  -159.990, Y  +432.766, Z    +0.000, E1  +383.321, E3 -418200.511}
SPL {X  -159.990, Y  +434.794, Z    +0.000, E1  +383.304, E3 -418210.543}
SPL {X  -159.990, Y  +437.007, Z    +0.000, E1  +383.323, E3 -418221.395}
SPL {X  -159.990, Y  +439.778, Z    +0.000, E1  +383.323, E3 -418235.027}
SPL {X  -159.990, Y  +442.945, Z    +0.000, E1  +383.339, E3 -418250.591}
SPL {X  -159.990, Y  +446.037, Z    +0.000, E1  +383.324, E3 -418265.842}
SPL {X  -159.990, Y  +448.341, Z    +0.000, E1  +383.317, E3 -418277.159}
SPL {X  -159.990, Y  +450.345, Z    +0.000, E1  +383.316, E3 -418287.037}
SPL {X  -159.990, Y  +452.828, Z    +0.000, E1  +383.330, E3 -418299.237}
SPL {X  -159.990, Y  +455.244, Z    +0.000, E1  +383.317, E3 -418311.136}
SPL {X  -159.990, Y  +457.167, Z    +0.000, E1  +383.324, E3 -418320.567}
SPL {X  -159.990, Y  +459.480, Z    +0.000, E1  +383.323, E3 -418331.970}
SPL {X  -159.990, Y  +462.520, Z    +0.000, E1  +383.350, E3 -418346.875}
SPL {X  -159.990, Y  +465.602, Z    +0.000, E1  +383.328, E3 -418362.074}
SPL {X  -159.990, Y  +467.934, Z    +0.000, E1  +383.321, E3 -418373.569}
SPL {X  -159.990, Y  +469.939, Z    +0.000, E1  +383.319, E3 -418383.430}
SPL {X  -159.990, Y  +472.144, Z    +0.000, E1  +383.327, E3 -418394.281}
SPL {X  -159.990, Y  +474.152, Z    +0.000, E1  +383.309, E3 -418404.233}
SPL {X  -159.990, Y  +476.560, Z    +0.000, E1  +383.332, E3 -418416.041}
SPL {X  -159.990, Y  +478.770, Z    +0.000, E1  +383.306, E3 -418426.966}
SPL {X  -159.990, Y  +480.905, Z    +0.000, E1  +383.327, E3 -418437.434}
SPL {X  -159.990, Y  +484.251, Z    +0.000, E1  +383.352, E3 -418453.850}
SPL {X  -159.990, Y  +488.031, Z    +0.000, E1  +383.345, E3 -418472.483}
SPL {X  -159.990, Y  +491.121, Z    +0.000, E1  +383.323, E3 -418487.728}
SPL {X  -159.990, Y  +493.610, Z    +0.000, E1  +383.323, E3 -418499.981}
SPL {X  -159.990, Y  +496.863, Z    +0.000, E1  +383.350, E3 -418515.941}
SPL {X  -159.990, Y  +499.995, Z    +0.000, E1  +383.324, E3 -418531.402}
SPL {X  -159.990, Y  +502.341, Z    +0.000, E1  +383.320, E3 -418542.962}
SPL {X  -159.990, Y  +505.377, Z    +0.000, E1  +383.346, E3 -418557.852}
SPL {X  -159.990, Y  +508.024, Z    +0.000, E1  +383.315, E3 -418570.934}
SPL {X  -159.990, Y  +510.344, Z    +0.000, E1  +383.327, E3 -418582.341}
SPL {X  -159.990, Y  +513.289, Z    +0.000, E1  +383.332, E3 -418596.831}
SPL {X  -159.990, Y  +516.195, Z    +0.000, E1  +383.325, E3 -418611.150}
SPL {X  -159.990, Y  +518.925, Z    +0.000, E1  +383.333, E3 -418624.514}
SPL {X  -159.990, Y  +521.408, Z    +0.000, E1  +383.329, E3 -418636.723}
SPL {X  -159.990, Y  +523.942, Z    +0.000, E1  +383.333, E3 -418649.215}
SPL {X  -159.990, Y  +526.221, Z    +0.000, E1  +383.314, E3 -418660.491}
SPL {X  -159.990, Y  +527.834, Z    +0.000, E1  +383.311, E3 -418668.441}
SPL {X  -159.990, Y  +529.993, Z    +0.000, E1  +383.329, E3 -418679.017}
SPL {X  -159.990, Y  +532.441, Z    +0.000, E1  +383.322, E3 -418691.068}
SPL {X  -159.990, Y  +534.618, Z    +0.000, E1  +383.322, E3 -418701.801}
SPL {X  -159.990, Y  +537.024, Z    +0.000, E1  +383.321, E3 -418713.663}
SPL {X  -159.990, Y  +539.129, Z    +0.000, E1  +383.310, E3 -418724.046}
SPL {X  -159.990, Y  +541.183, Z    +0.000, E1  +383.319, E3 -418734.143}
SPL {X  -159.990, Y  +543.647, Z    +0.000, E1  +383.325, E3 -418746.246}
SPL {X  -159.990, Y  +546.832, Z    +0.000, E1  +383.349, E3 -418761.869}
SPL {X  -159.990, Y  +549.756, Z    +0.000, E1  +383.320, E3 -418776.310}
SPL {X  -159.990, Y  +551.655, Z    +0.000, E1  +383.320, E3 -418785.661}
SPL {X  -159.990, Y  +553.711, Z    +0.000, E1  +383.317, E3 -418795.783}
SPL {X  -159.990, Y  +555.637, Z    +0.000, E1  +383.323, E3 -418805.251}
SPL {X  -159.990, Y  +558.758, Z    +0.000, E1  +383.351, E3 -418820.561}
SPL {X  -159.990, Y  +561.830, Z    +0.000, E1  +383.325, E3 -418835.734}
SPL {X  -159.990, Y  +564.273, Z    +0.000, E1  +383.325, E3 -418847.759}
SPL {X  -159.990, Y  +567.351, Z    +0.000, E1  +383.348, E3 -418862.854}
SPL {X  -159.990, Y  +570.314, Z    +0.000, E1  +383.326, E3 -418877.486}
SPL {X  -159.990, Y  +572.504, Z    +0.000, E1  +383.321, E3 -418888.271}
SPL {X  -159.990, Y  +575.653, Z    +0.000, E1  +383.355, E3 -418903.708}
SPL {X  -159.990, Y  +578.932, Z    +0.000, E1  +383.330, E3 -418919.891}
SPL {X  -159.990, Y  +581.497, Z    +0.000, E1  +383.329, E3 -418932.476}
SPL {X  -159.990, Y  +583.973, Z    +0.000, E1  +383.332, E3 -418944.661}
SPL {X  -159.990, Y  +586.877, Z    +0.000, E1  +383.349, E3 -418958.915}
SPL {X  -159.990, Y  +590.594, Z    +0.000, E1  +383.363, E3 -418977.166}
SPL {X  -159.990, Y  +593.847, Z    +0.000, E1  +383.340, E3 -418993.176}
SPL {X  -159.990, Y  +597.018, Z    +0.000, E1  +383.367, E3 -419008.708}
SPL {X  -159.990, Y  +599.887, Z    +0.000, E1  +383.341, E3 -419022.812}
SPL {X  -159.990, Y  +601.949, Z    +0.000, E1  +383.344, E3 -419032.939}
SPL {X  -159.990, Y  +605.106, Z    +0.000, E1  +383.383, E3 -419048.385}
SPL {X  -159.990, Y  +608.111, Z    +0.000, E1  +383.342, E3 -419063.236}
SPL {X  -159.990, Y  +610.073, Z    +0.000, E1  +383.343, E3 -419072.894}
SPL {X  -159.990, Y  +613.021, Z    +0.000, E1  +383.365, E3 -419087.364}
SPL {X  -159.990, Y  +615.657, Z    +0.000, E1  +383.331, E3 -419100.413}
SPL {X  -159.990, Y  +617.658, Z    +0.000, E1  +383.335, E3 -419110.255}
SPL {X  -159.990, Y  +620.788, Z    +0.000, E1  +383.368, E3 -419125.588}
SPL {X  -159.990, Y  +624.347, Z    +0.000, E1  +383.355, E3 -419143.108}
SPL {X  -159.990, Y  +627.144, Z    +0.000, E1  +383.340, E3 -419156.878}
SPL {X  -159.990, Y  +629.284, Z    +0.000, E1  +383.339, E3 -419167.385}
SPL {X  -159.990, Y  +631.206, Z    +0.000, E1  +383.337, E3 -419176.839}
SPL {X  -159.990, Y  +633.318, Z    +0.000, E1  +383.339, E3 -419187.244}
SPL {X  -159.990, Y  +635.650, Z    +0.000, E1  +383.339, E3 -419198.714}
SPL {X  -159.990, Y  +637.597, Z    +0.000, E1  +383.330, E3 -419208.337}
SPL {X  -159.990, Y  +640.369, Z    +0.000, E1  +383.354, E3 -419221.971}
SPL {X  -159.990, Y  +644.241, Z    +0.000, E1  +383.355, E3 -419241.083}
SPL {X  -159.990, Y  +648.287, Z    +0.000, E1  +383.349, E3 -419261.040}
SPL {X  -159.990, Y  +651.427, Z    +0.000, E1  +383.319, E3 -419276.535}
SPL {X  -159.990, Y  +653.536, Z    +0.000, E1  +383.313, E3 -419286.917}
SPL {X  -159.990, Y  +656.380, Z    +0.000, E1  +383.347, E3 -419300.853}
SPL {X  -159.990, Y  +659.180, Z    +0.000, E1  +383.314, E3 -419314.701}
SPL {X  -159.990, Y  +661.392, Z    +0.000, E1  +383.318, E3 -419325.594}
SPL {X  -159.990, Y  +663.662, Z    +0.000, E1  +383.322, E3 -419336.718}
SPL {X  -159.990, Y  +665.964, Z    +0.000, E1  +383.328, E3 -419348.009}
SPL {X  -159.990, Y  +668.989, Z    +0.000, E1  +383.359, E3 -419362.845}
SPL {X  -159.983, Y  +672.946, Z    +0.000, E1  +383.359, E3 -419382.326}
SPL {X  -159.924, Y  +676.110, Z    +0.000, E1  +383.320, E3 -419398.025}
SPL {X  -159.845, Y  +678.302, Z    +0.000, E1  +383.298, E3 -419408.927}
SPL {X  -159.760, Y  +680.081, Z    +0.000, E1  +383.288, E3 -419417.771}
SPL {X  -159.626, Y  +682.287, Z    +0.000, E1  +383.280, E3 -419428.742}
SPL {X  -159.462, Y  +684.486, Z    +0.000, E1  +383.258, E3 -419439.742}
SPL {X  -159.212, Y  +687.262, Z    +0.000, E1  +383.238, E3 -419453.646}
SPL {X  -158.971, Y  +689.529, Z    +0.000, E1  +383.181, E3 -419465.106}
SPL {X  -158.658, Y  +692.098, Z    +0.000, E1  +383.176, E3 -419478.012}
ENDSPLINE

SPLINE
SPL {X  -159.063, Y  +688.696, Z    +0.000, E1  +377.094, E3 -419520.231}
SPL {X  -159.987, Y  +672.488, Z    +0.000, E1  +365.638, E3 -419544.296}
SPL {X  -159.990, Y  +663.928, Z    +0.000, E1  +359.662, E3 -419550.090}
SPL {X  -159.990, Y  +658.009, Z    +0.000, E1  +355.226, E3 -419553.790}
SPL {X  -159.990, Y  +651.879, Z    +0.000, E1  +350.548, E3 -419558.853}
SPL {X  -159.990, Y  +637.832, Z    +0.000, E1  +341.694, E3 -419576.444}
SPL {X  -159.990, Y  +626.634, Z    +0.000, E1  +337.968, E3 -419607.297}
SPL {X  -159.990, Y  +624.622, Z    +0.000, E1  +337.980, E3 -419617.881}
SPL {X  -159.990, Y  +622.489, Z    +0.000, E1  +337.969, E3 -419629.047}
SPL {X  -159.990, Y  +619.955, Z    +0.000, E1  +337.968, E3 -419642.337}
SPL {X  -159.990, Y  +617.386, Z    +0.000, E1  +337.968, E3 -419655.812}
SPL {X  -159.990, Y  +614.863, Z    +0.000, E1  +337.969, E3 -419669.044}
SPL {X  -159.990, Y  +612.600, Z    +0.000, E1  +337.975, E3 -419680.928}
SPL {X  -159.990, Y  +610.646, Z    +0.000, E1  +337.979, E3 -419691.185}
SPL {X  -159.990, Y  +608.810, Z    +0.000, E1  +337.977, E3 -419700.818}
SPL {X  -159.990, Y  +605.804, Z    +0.000, E1  +337.936, E3 -419716.464}
SPL {X  -159.990, Y  +602.819, Z    +0.000, E1  +337.963, E3 -419732.135}
SPL {X  -159.990, Y  +600.642, Z    +0.000, E1  +337.968, E3 -419743.563}
SPL {X  -159.990, Y  +598.568, Z    +0.000, E1  +337.954, E3 -419754.356}
SPL {X  -159.990, Y  +596.440, Z    +0.000, E1  +337.964, E3 -419765.537}
SPL {X  -159.990, Y  +593.768, Z    +0.000, E1  +337.929, E3 -419779.470}
SPL {X  -159.990, Y  +590.068, Z    +0.000, E1  +337.924, E3 -419798.838}
SPL {X  -159.990, Y  +586.620, Z    +0.000, E1  +337.935, E3 -419816.901}
SPL {X  -159.990, Y  +584.080, Z    +0.000, E1  +337.953, E3 -419830.227}
SPL {X  -159.990, Y  +581.924, Z    +0.000, E1  +337.949, E3 -419841.528}
SPL {X  -159.990, Y  +578.886, Z    +0.000, E1  +337.918, E3 -419857.382}
SPL {X  -159.990, Y  +576.252, Z    +0.000, E1  +337.962, E3 -419871.280}
SPL {X  -159.990, Y  +574.188, Z    +0.000, E1  +337.947, E3 -419882.053}
SPL {X  -159.990, Y  +571.954, Z    +0.000, E1  +337.959, E3 -419893.810}
SPL {X  -159.990, Y  +570.110, Z    +0.000, E1  +337.958, E3 -419903.461}
SPL {X  -159.990, Y  +568.165, Z    +0.000, E1  +337.957, E3 -419913.640}
SPL {X  -159.990, Y  +566.106, Z    +0.000, E1  +337.954, E3 -419924.424}
SPL {X  -159.990, Y  +563.259, Z    +0.000, E1  +337.929, E3 -419939.306}
SPL {X  -159.990, Y  +559.661, Z    +0.000, E1  +337.922, E3 -419958.128}
SPL {X  -159.990, Y  +555.965, Z    +0.000, E1  +337.915, E3 -419977.437}
SPL {X  -159.990, Y  +553.115, Z    +0.000, E1  +337.946, E3 -419992.423}
SPL {X  -159.990, Y  +550.886, Z    +0.000, E1  +337.944, E3 -420004.104}
SPL {X  -159.990, Y  +548.568, Z    +0.000, E1  +337.944, E3 -420016.225}
SPL {X  -159.990, Y  +546.537, Z    +0.000, E1  +337.948, E3 -420026.860}
SPL {X  -159.990, Y  +545.062, Z    +0.000, E1  +337.955, E3 -420034.619}
SPL {X  -159.990, Y  +543.060, Z    +0.000, E1  +337.943, E3 -420045.098}
SPL {X  -159.990, Y  +539.928, Z    +0.000, E1  +337.917, E3 -420061.440}
SPL {X  -159.990, Y  +536.935, Z    +0.000, E1  +337.942, E3 -420077.157}
SPL {X  -159.990, Y  +534.656, Z    +0.000, E1  +337.946, E3 -420089.100}
SPL {X  -159.990, Y  +531.679, Z    +0.000, E1  +337.913, E3 -420104.614}
SPL {X  -159.990, Y  +527.941, Z    +0.000, E1  +337.907, E3 -420124.156}
SPL {X  -159.990, Y  +525.053, Z    +0.000, E1  +337.942, E3 -420139.347}
SPL {X  -159.990, Y  +522.838, Z    +0.000, E1  +337.933, E3 -420150.951}
SPL {X  -159.990, Y  +519.698, Z    +0.000, E1  +337.916, E3 -420167.334}
SPL {X  -159.990, Y  +517.251, Z    +0.000, E1  +337.946, E3 -420180.194}
SPL {X  -159.990, Y  +515.568, Z    +0.000, E1  +338.084, E3 -420190.291}
ENDSPLINE

SPLINE
SPL {X  -159.990, Y  +518.374, Z    +0.000, E1  +341.240, E3 -420202.878}
ENDSPLINE

SPLINE
SPL {X  -159.990, Y  +513.606, Z    +0.000, E1  +339.879, E3 -420218.789}
SPL {X  -159.990, Y  +508.660, Z    +0.000, E1  +338.515, E3 -420234.219}
SPL {X  -159.990, Y  +505.237, Z    +0.000, E1  +337.606, E3 -420244.476}
SPL {X  -159.990, Y  +501.963, Z    +0.000, E1  +336.712, E3 -420253.580}
SPL {X  -159.990, Y  +498.406, Z    +0.000, E1  +335.789, E3 -420263.331}
SPL {X  -159.990, Y  +494.693, Z    +0.000, E1  +334.929, E3 -420273.798}
SPL {X  -159.990, Y  +491.649, Z    +0.000, E1  +334.596, E3 -420285.001}
SPL {X  -159.990, Y  +488.807, Z    +0.000, E1  +334.603, E3 -420297.725}
SPL {X  -159.990, Y  +486.070, Z    +0.000, E1  +334.601, E3 -420309.956}
SPL {X  -159.990, Y  +482.821, Z    +0.000, E1  +334.589, E3 -420324.457}
SPL {X  -159.990, Y  +480.183, Z    +0.000, E1  +334.616, E3 -420336.298}
SPL {X  -159.990, Y  +477.508, Z    +0.000, E1  +334.590, E3 -420348.206}
SPL {X  -159.990, Y  +473.634, Z    +0.000, E1  +334.574, E3 -420365.495}
SPL {X  -159.990, Y  +470.047, Z    +0.000, E1  +334.598, E3 -420381.576}
SPL {X  -159.990, Y  +467.082, Z    +0.000, E1  +334.601, E3 -420394.824}
SPL {X  -159.990, Y  +464.063, Z    +0.000, E1  +334.595, E3 -420408.319}
SPL {X  -159.990, Y  +460.712, Z    +0.000, E1  +334.589, E3 -420423.278}
SPL {X  -159.990, Y  +457.497, Z    +0.000, E1  +334.597, E3 -420437.651}
SPL {X  -159.990, Y  +454.323, Z    +0.000, E1  +334.588, E3 -420451.810}
SPL {X  -159.990, Y  +450.823, Z    +0.000, E1  +334.583, E3 -420467.439}
SPL {X  -159.990, Y  +447.982, Z    +0.000, E1  +334.607, E3 -420480.179}
SPL {X  -159.990, Y  +445.108, Z    +0.000, E1  +334.593, E3 -420493.056}
SPL {X  -159.990, Y  +441.797, Z    +0.000, E1  +334.610, E3 -420507.935}
SPL {X  -159.990, Y  +439.442, Z    +0.000, E1  +334.631, E3 -420518.512}
SPL {X  -159.990, Y  +436.316, Z    +0.000, E1  +334.580, E3 -420532.394}
SPL {X  -159.990, Y  +432.613, Z    +0.000, E1  +334.610, E3 -420549.020}
SPL {X  -159.990, Y  +429.827, Z    +0.000, E1  +334.620, E3 -420561.497}
SPL {X  -159.990, Y  +426.865, Z    +0.000, E1  +334.602, E3 -420574.702}
SPL {X  -159.990, Y  +423.417, Z    +0.000, E1  +334.600, E3 -420590.118}
SPL {X  -159.990, Y  +420.283, Z    +0.000, E1  +334.614, E3 -420604.162}
SPL {X  -159.990, Y  +417.103, Z    +0.000, E1  +334.600, E3 -420618.357}
SPL {X  -159.990, Y  +413.684, Z    +0.000, E1  +334.603, E3 -420633.656}
SPL {X  -159.990, Y  +410.645, Z    +0.000, E1  +334.615, E3 -420647.268}
SPL {X  -159.990, Y  +407.450, Z    +0.000, E1  +334.599, E3 -420661.517}
SPL {X  -159.990, Y  +403.513, Z    +0.000, E1  +334.580, E3 -420679.070}
SPL {X  -159.990, Y  +400.403, Z    +0.000, E1  +334.620, E3 -420693.053}
SPL {X  -159.990, Y  +397.743, Z    +0.000, E1  +334.600, E3 -420704.922}
SPL {X  -159.990, Y  +394.848, Z    +0.000, E1  +334.621, E3 -420717.923}
SPL {X  -159.990, Y  +392.473, Z    +0.000, E1  +334.623, E3 -420728.550}
SPL {X  -159.990, Y  +390.187, Z    +0.000, E1  +334.622, E3 -420738.808}
SPL {X  -159.990, Y  +387.503, Z    +0.000, E1  +334.622, E3 -420750.803}
SPL {X  -159.990, Y  +384.711, Z    +0.000, E1  +334.612, E3 -420763.246}
SPL {X  -159.988, Y  +381.794, Z    +0.000, E1  +334.611, E3 -420776.281}
SPL {X  -159.958, Y  +379.279, Z    +0.000, E1  +334.625, E3 -420787.571}
SPL {X  -159.894, Y  +376.959, Z    +0.000, E1  +334.630, E3 -420798.016}
SPL {X  -159.765, Y  +374.027, Z    +0.000, E1  +334.633, E3 -420811.231}
SPL {X  -159.607, Y  +371.442, Z    +0.000, E1  +334.673, E3 -420823.006}
SPL {X  -159.379, Y  +368.534, Z    +0.000, E1  +334.684, E3 -420836.194}
SPL {X  -159.113, Y  +365.767, Z    +0.000, E1  +334.734, E3 -420848.833}
SPL {X  -158.798, Y  +363.007, Z    +0.000, E1  +334.761, E3 -420861.474}
SPL {X  -158.453, Y  +360.380, Z    +0.000, E1  +334.828, E3 -420873.618}
SPL {X  -158.127, Y  +358.155, Z    +0.000, E1  +334.874, E3 -420883.949}
SPL {X  -158.095, Y  +357.947, Z    +0.000, E1  +338.259, E3 -420915.521}
ENDSPLINE

SPLINE
SPL {X  -158.454, Y  +360.384, Z    +0.000, E1  +340.634, E3 -420927.672}
SPL {X  -159.737, Y  +373.507, Z    +0.000, E1  +349.689, E3 -420949.708}
SPL {X  -159.990, Y  +382.574, Z    +0.000, E1  +355.537, E3 -420956.396}
SPL {X  -159.990, Y  +389.909, Z    +0.000, E1  +360.662, E3 -420960.410}
SPL {X  -159.990, Y  +396.289, Z    +0.000, E1  +365.500, E3 -420964.190}
SPL {X  -159.990, Y  +407.941, Z    +0.000, E1  +374.126, E3 -420975.527}
SPL {X  -159.990, Y  +418.671, Z    +0.000, E1  +379.855, E3 -420994.943}
SPL {X  -159.990, Y  +429.878, Z    +0.000, E1  +383.330, E3 -421024.998}
SPL {X  -159.990, Y  +432.103, Z    +0.000, E1  +383.301, E3 -421036.017}
SPL {X  -159.990, Y  +434.188, Z    +0.000, E1  +383.325, E3 -421046.214}
SPL {X  -159.990, Y  +436.320, Z    +0.000, E1  +383.304, E3 -421056.766}
SPL {X  -159.990, Y  +439.169, Z    +0.000, E1  +383.353, E3 -421070.683}
SPL {X  -159.990, Y  +442.945, Z    +0.000, E1  +383.339, E3 -421089.301}
SPL {X  -159.990, Y  +446.037, Z    +0.000, E1  +383.324, E3 -421104.551}
SPL {X  -159.990, Y  +448.341, Z    +0.000, E1  +383.317, E3 -421115.869}
SPL {X  -159.990, Y  +450.345, Z    +0.000, E1  +383.316, E3 -421125.747}
SPL {X  -159.990, Y  +452.828, Z    +0.000, E1  +383.330, E3 -421137.946}
SPL {X  -159.990, Y  +456.338, Z    +0.000, E1  +383.359, E3 -421155.138}
SPL {X  -159.990, Y  +459.480, Z    +0.000, E1  +383.323, E3 -421170.680}
SPL {X  -159.990, Y  +461.803, Z    +0.000, E1  +383.322, E3 -421182.115}
SPL {X  -159.990, Y  +464.971, Z    +0.000, E1  +383.357, E3 -421197.621}
SPL {X  -159.990, Y  +467.934, Z    +0.000, E1  +383.321, E3 -421212.278}
SPL {X  -159.990, Y  +469.939, Z    +0.000, E1  +383.319, E3 -421222.140}
SPL {X  -159.990, Y  +472.144, Z    +0.000, E1  +383.327, E3 -421232.991}
SPL {X  -159.990, Y  +474.994, Z    +0.000, E1  +383.334, E3 -421247.039}
SPL {X  -159.990, Y  +477.323, Z    +0.000, E1  +383.307, E3 -421258.554}
SPL {X  -159.990, Y  +479.553, Z    +0.000, E1  +383.328, E3 -421269.489}
SPL {X  -159.990, Y  +482.799, Z    +0.000, E1  +383.343, E3 -421285.429}
SPL {X  -159.990, Y  +485.299, Z    +0.000, E1  +383.310, E3 -421297.814}
SPL {X  -159.990, Y  +488.031, Z    +0.000, E1  +383.345, E3 -421311.192}
SPL {X  -159.990, Y  +491.121, Z    +0.000, E1  +383.323, E3 -421326.438}
SPL {X  -159.990, Y  +493.610, Z    +0.000, E1  +383.323, E3 -421338.691}
SPL {X  -159.990, Y  +495.794, Z    +0.000, E1  +383.312, E3 -421349.464}
SPL {X  -159.990, Y  +497.668, Z    +0.000, E1  +383.317, E3 -421358.674}
SPL {X  -159.990, Y  +499.995, Z    +0.000, E1  +383.324, E3 -421370.112}
SPL {X  -159.990, Y  +502.341, Z    +0.000, E1  +383.320, E3 -421381.671}
SPL {X  -159.990, Y  +504.419, Z    +0.000, E1  +383.313, E3 -421391.913}
SPL {X  -159.990, Y  +507.187, Z    +0.000, E1  +383.346, E3 -421405.466}
SPL {X  -159.990, Y  +510.344, Z    +0.000, E1  +383.327, E3 -421421.051}
SPL {X  -159.990, Y  +512.484, Z    +0.000, E1  +383.309, E3 -421431.623}
SPL {X  -159.990, Y  +514.016, Z    +0.000, E1  +383.308, E3 -421439.172}
SPL {X  -159.990, Y  +516.195, Z    +0.000, E1  +383.325, E3 -421449.860}
SPL {X  -159.990, Y  +518.925, Z    +0.000, E1  +383.333, E3 -421463.223}
SPL {X  -159.990, Y  +521.408, Z    +0.000, E1  +383.329, E3 -421475.432}
SPL {X  -159.990, Y  +523.942, Z    +0.000, E1  +383.333, E3 -421487.925}
SPL {X  -159.990, Y  +526.221, Z    +0.000, E1  +383.314, E3 -421499.201}
SPL {X  -159.990, Y  +527.834, Z    +0.000, E1  +383.311, E3 -421507.151}
SPL {X  -159.990, Y  +529.993, Z    +0.000, E1  +383.329, E3 -421517.727}
SPL {X  -159.990, Y  +532.441, Z    +0.000, E1  +383.322, E3 -421529.778}
SPL {X  -159.990, Y  +534.618, Z    +0.000, E1  +383.322, E3 -421540.511}
SPL {X  -159.990, Y  +537.024, Z    +0.000, E1  +383.321, E3 -421552.373}
SPL {X  -159.990, Y  +539.129, Z    +0.000, E1  +383.310, E3 -421562.756}
SPL {X  -159.990, Y  +541.183, Z    +0.000, E1  +383.319, E3 -421572.853}
SPL {X  -159.990, Y  +543.647, Z    +0.000, E1  +383.325, E3 -421584.956}
SPL {X  -159.990, Y  +545.957, Z    +0.000, E1  +383.318, E3 -421596.336}
SPL {X  -159.990, Y  +548.912, Z    +0.000, E1  +383.354, E3 -421610.795}
SPL {X  -159.990, Y  +551.655, Z    +0.000, E1  +383.320, E3 -421624.370}
SPL {X  -159.990, Y  +553.711, Z    +0.000, E1  +383.317, E3 -421634.492}
SPL {X  -159.990, Y  +556.481, Z    +0.000, E1  +383.354, E3 -421648.054}
SPL {X  -159.990, Y  +559.475, Z    +0.000, E1  +383.321, E3 -421662.859}
SPL {X  -159.990, Y  +561.830, Z    +0.000, E1  +383.325, E3 -421674.444}
SPL {X  -159.990, Y  +564.273, Z    +0.000, E1  +383.325, E3 -421686.468}
SPL {X  -159.990, Y  +566.342, Z    +0.000, E1  +383.314, E3 -421696.673}
SPL {X  -159.990, Y  +568.184, Z    +0.000, E1  +383.317, E3 -421705.734}
SPL {X  -159.990, Y  +570.314, Z    +0.000, E1  +383.326, E3 -421716.196}
SPL {X  -159.990, Y  +573.444, Z    +0.000, E1  +383.356, E3 -421731.535}
SPL {X  -159.990, Y  +577.161, Z    +0.000, E1  +383.346, E3 -421749.860}
SPL {X  -159.990, Y  +580.840, Z    +0.000, E1  +383.355, E3 -421767.909}
SPL {X  -159.990, Y  +583.973, Z    +0.000, E1  +383.332, E3 -421783.370}
SPL {X  -159.990, Y  +586.020, Z    +0.000, E1  +383.323, E3 -421793.454}
SPL {X  -159.990, Y  +587.711, Z    +0.000, E1  +383.318, E3 -421801.794}
SPL {X  -159.990, Y  +589.763, Z    +0.000, E1  +383.328, E3 -421811.870}
SPL {X  -159.990, Y  +591.698, Z    +0.000, E1  +383.324, E3 -421821.355}
SPL {X  -159.990, Y  +593.847, Z    +0.000, E1  +383.340, E3 -421831.886}
SPL {X  -159.990, Y  +597.018, Z    +0.000, E1  +383.367, E3 -421847.417}
SPL {X  -159.990, Y  +599.887, Z    +0.000, E1  +383.341, E3 -421861.522}
SPL {X  -159.990, Y  +601.949, Z    +0.000, E1  +383.344, E3 -421871.648}
SPL {X  -159.990, Y  +605.106, Z    +0.000, E1  +383.383, E3 -421887.095}
SPL {X  -159.990, Y  +608.111, Z    +0.000, E1  +383.342, E3 -421901.945}
SPL {X  -159.990, Y  +610.073, Z    +0.000, E1  +383.343, E3 -421911.603}
SPL {X  -159.990, Y  +612.330, Z    +0.000, E1  +383.340, E3 -421922.731}
SPL {X  -159.990, Y  +615.036, Z    +0.000, E1  +383.353, E3 -421936.018}
SPL {X  -159.990, Y  +618.481, Z    +0.000, E1  +383.366, E3 -421952.956}
SPL {X  -159.990, Y  +621.517, Z    +0.000, E1  +383.337, E3 -421967.939}
SPL {X  -159.990, Y  +623.764, Z    +0.000, E1  +383.335, E3 -421978.990}
SPL {X  -159.990, Y  +626.608, Z    +0.000, E1  +383.361, E3 -421992.915}
SPL {X  -159.990, Y  +630.271, Z    +0.000, E1  +383.375, E3 -422010.876}
SPL {X  -159.990, Y  +633.318, Z    +0.000, E1  +383.339, E3 -422025.953}
SPL {X  -159.990, Y  +635.650, Z    +0.000, E1  +383.339, E3 -422037.424}
SPL {X  -159.990, Y  +638.406, Z    +0.000, E1  +383.354, E3 -422050.991}
SPL {X  -159.990, Y  +641.831, Z    +0.000, E1  +383.342, E3 -422067.938}
SPL {X  -159.990, Y  +644.884, Z    +0.000, E1  +383.324, E3 -422083.025}
SPL {X  -159.990, Y  +647.550, Z    +0.000, E1  +383.318, E3 -422096.192}
SPL {X  -159.990, Y  +650.790, Z    +0.000, E1  +383.346, E3 -422112.059}
SPL {X  -159.990, Y  +654.543, Z    +0.000, E1  +383.348, E3 -422130.511}
SPL {X  -159.990, Y  +658.319, Z    +0.000, E1  +383.349, E3 -422149.101}
SPL {X  -159.990, Y  +661.392, Z    +0.000, E1  +383.318, E3 -422164.304}
SPL {X  -159.990, Y  +663.662, Z    +0.000, E1  +383.322, E3 -422175.428}
SPL {X  -159.990, Y  +665.964, Z    +0.000, E1  +383.328, E3 -422186.719}
SPL {X  -159.990, Y  +667.870, Z    +0.000, E1  +383.320, E3 -422196.126}
SPL {X  -159.990, Y  +669.861, Z    +0.000, E1  +383.321, E3 -422205.927}
SPL {X  -159.983, Y  +672.946, Z    +0.000, E1  +383.359, E3 -422221.036}
SPL {X  -159.924, Y  +676.110, Z    +0.000, E1  +383.320, E3 -422236.735}
SPL {X  -159.801, Y  +679.265, Z    +0.000, E1  +383.327, E3 -422252.354}
SPL {X  -159.626, Y  +682.287, Z    +0.000, E1  +383.280, E3 -422267.452}
SPL {X  -159.462, Y  +684.486, Z    +0.000, E1  +383.258, E3 -422278.452}
SPL {X  -159.289, Y  +686.457, Z    +0.000, E1  +383.223, E3 -422288.362}
SPL {X  -159.052, Y  +688.801, Z    +0.000, E1  +383.217, E3 -422300.096}
SPL {X  -158.770, Y  +691.222, Z    +0.000, E1  +383.158, E3 -422312.354}
SPL {X  -158.553, Y  +692.896, Z    +0.000, E1  +383.130, E3 -422320.820}
ENDSPLINE

SPLINE
SPL {X  -159.063, Y  +688.696, Z    +0.000, E1  +377.094, E3 -422358.941}
SPL {X  -159.987, Y  +672.488, Z    +0.000, E1  +365.638, E3 -422383.005}
SPL {X  -159.990, Y  +663.928, Z    +0.000, E1  +359.662, E3 -422388.800}
SPL {X  -159.990, Y  +658.009, Z    +0.000, E1  +355.226, E3 -422392.500}
SPL {X  -159.990, Y  +651.879, Z    +0.000, E1  +350.548, E3 -422397.562}
SPL {X  -159.990, Y  +637.832, Z    +0.000, E1  +341.694, E3 -422415.153}
SPL {X  -159.990, Y  +626.634, Z    +0.000, E1  +337.968, E3 -422446.007}
SPL {X  -159.990, Y  +624.622, Z    +0.000, E1  +337.980, E3 -422456.590}
SPL {X  -159.990, Y  +622.489, Z    +0.000, E1  +337.969, E3 -422467.757}
SPL {X  -159.990, Y  +619.955, Z    +0.000, E1  +337.968, E3 -422481.047}
SPL {X  -159.990, Y  +617.386, Z    +0.000, E1  +337.968, E3 -422494.521}
SPL {X  -159.990, Y  +614.863, Z    +0.000, E1  +337.969, E3 -422507.754}
SPL {X  -159.990, Y  +612.600, Z    +0.000, E1  +337.975, E3 -422519.638}
SPL {X  -159.990, Y  +610.646, Z    +0.000, E1  +337.979, E3 -422529.895}
SPL {X  -159.990, Y  +608.810, Z    +0.000, E1  +337.977, E3 -422539.528}
SPL {X  -159.990, Y  +606.481, Z    +0.000, E1  +337.967, E3 -422551.703}
SPL {X  -159.990, Y  +603.419, Z    +0.000, E1  +337.936, E3 -422567.643}
SPL {X  -159.990, Y  +600.642, Z    +0.000, E1  +337.968, E3 -422582.273}
SPL {X  -159.990, Y  +598.568, Z    +0.000, E1  +337.954, E3 -422593.065}
SPL {X  -159.990, Y  +595.493, Z    +0.000, E1  +337.930, E3 -422609.149}
SPL {X  -159.990, Y  +592.865, Z    +0.000, E1  +337.964, E3 -422622.977}
SPL {X  -159.990, Y  +590.803, Z    +0.000, E1  +337.954, E3 -422633.768}
SPL {X  -159.990, Y  +588.288, Z    +0.000, E1  +337.950, E3 -422646.932}
SPL {X  -159.990, Y  +586.040, Z    +0.000, E1  +337.954, E3 -422658.677}
SPL {X  -159.990, Y  +584.080, Z    +0.000, E1  +337.953, E3 -422668.937}
SPL {X  -159.990, Y  +581.924, Z    +0.000, E1  +337.949, E3 -422680.237}
SPL {X  -159.990, Y  +579.673, Z    +0.000, E1  +337.950, E3 -422692.036}
SPL {X  -159.990, Y  +576.961, Z    +0.000, E1  +337.936, E3 -422706.215}
SPL {X  -159.990, Y  +574.188, Z    +0.000, E1  +337.947, E3 -422720.762}
SPL {X  -159.990, Y  +571.954, Z    +0.000, E1  +337.959, E3 -422732.520}
SPL {X  -159.990, Y  +570.110, Z    +0.000, E1  +337.958, E3 -422742.170}
SPL {X  -159.990, Y  +568.165, Z    +0.000, E1  +337.957, E3 -422752.350}
SPL {X  -159.990, Y  +565.292, Z    +0.000, E1  +337.922, E3 -422767.328}
SPL {X  -159.990, Y  +562.598, Z    +0.000, E1  +337.958, E3 -422781.539}
SPL {X  -159.990, Y  +560.652, Z    +0.000, E1  +337.962, E3 -422791.751}
SPL {X  -159.990, Y  +558.143, Z    +0.000, E1  +337.928, E3 -422804.783}
SPL {X  -159.990, Y  +555.329, Z    +0.000, E1  +337.943, E3 -422819.527}
SPL {X  -159.990, Y  +553.115, Z    +0.000, E1  +337.946, E3 -422831.132}
SPL {X  -159.990, Y  +550.886, Z    +0.000, E1  +337.944, E3 -422842.814}
SPL {X  -159.990, Y  +548.568, Z    +0.000, E1  +337.944, E3 -422854.935}
SPL {X  -159.990, Y  +545.859, Z    +0.000, E1  +337.926, E3 -422869.084}
SPL {X  -159.990, Y  +542.390, Z    +0.000, E1  +337.914, E3 -422887.255}
SPL {X  -159.990, Y  +539.341, Z    +0.000, E1  +337.944, E3 -422903.276}
SPL {X  -159.990, Y  +536.935, Z    +0.000, E1  +337.942, E3 -422915.866}
SPL {X  -159.990, Y  +534.656, Z    +0.000, E1  +337.946, E3 -422927.810}
SPL {X  -159.990, Y  +532.453, Z    +0.000, E1  +337.944, E3 -422939.337}
SPL {X  -159.990, Y  +530.660, Z    +0.000, E1  +337.952, E3 -422948.739}
SPL {X  -159.990, Y  +528.702, Z    +0.000, E1  +337.939, E3 -422958.953}
SPL {X  -159.990, Y  +525.760, Z    +0.000, E1  +337.914, E3 -422974.294}
SPL {X  -159.990, Y  +522.838, Z    +0.000, E1  +337.933, E3 -422989.661}
SPL {X  -159.990, Y  +519.698, Z    +0.000, E1  +337.916, E3 -423006.044}
SPL {X  -159.990, Y  +517.251, Z    +0.000, E1  +337.946, E3 -423018.903}
SPL {X  -159.990, Y  +515.568, Z    +0.000, E1  +338.084, E3 -423029.000}
ENDSPLINE

SPLINE
SPL {X  -159.990, Y  +517.293, Z    +0.000, E1  +340.923, E3 -423045.299}
ENDSPLINE

SPLINE
SPL {X  -159.990, Y  +512.548, Z    +0.000, E1  +339.587, E3 -423060.874}
SPL {X  -159.990, Y  +508.660, Z    +0.000, E1  +338.515, E3 -423072.928}
SPL {X  -159.990, Y  +503.499, Z    +0.000, E1  +337.116, E3 -423088.007}
SPL {X  -159.990, Y  +498.406, Z    +0.000, E1  +335.789, E3 -423102.040}
SPL {X  -159.990, Y  +494.693, Z    +0.000, E1  +334.929, E3 -423112.508}
SPL {X  -159.990, Y  +491.649, Z    +0.000, E1  +334.596, E3 -423123.710}
SPL {X  -159.990, Y  +488.807, Z    +0.000, E1  +334.603, E3 -423136.435}
SPL {X  -159.990, Y  +486.070, Z    +0.000, E1  +334.601, E3 -423148.666}
SPL {X  -159.990, Y  +483.747, Z    +0.000, E1  +334.616, E3 -423159.078}
SPL {X  -159.990, Y  +481.038, Z    +0.000, E1  +334.588, E3 -423171.134}
SPL {X  -159.990, Y  +478.407, Z    +0.000, E1  +334.616, E3 -423182.948}
SPL {X  -159.990, Y  +475.940, Z    +0.000, E1  +334.597, E3 -423193.938}
SPL {X  -159.990, Y  +473.026, Z    +0.000, E1  +334.601, E3 -423206.968}
SPL {X  -159.990, Y  +470.047, Z    +0.000, E1  +334.598, E3 -423220.286}
SPL {X  -159.990, Y  +467.082, Z    +0.000, E1  +334.601, E3 -423233.533}
SPL {X  -159.990, Y  +464.919, Z    +0.000, E1  +334.619, E3 -423243.260}
SPL {X  -159.990, Y  +462.520, Z    +0.000, E1  +334.600, E3 -423253.934}
SPL {X  -159.990, Y  +460.081, Z    +0.000, E1  +334.610, E3 -423264.836}
SPL {X  -159.990, Y  +457.497, Z    +0.000, E1  +334.597, E3 -423276.360}
SPL {X  -159.990, Y  +454.323, Z    +0.000, E1  +334.588, E3 -423290.519}
SPL {X  -159.990, Y  +450.823, Z    +0.000, E1  +334.583, E3 -423306.148}
SPL {X  -159.990, Y  +446.894, Z    +0.000, E1  +334.572, E3 -423323.705}
SPL {X  -159.990, Y  +443.345, Z    +0.000, E1  +334.610, E3 -423339.713}
SPL {X  -159.990, Y  +441.077, Z    +0.000, E1  +334.631, E3 -423349.911}
SPL {X  -159.990, Y  +438.608, Z    +0.000, E1  +334.608, E3 -423360.908}
SPL {X  -159.990, Y  +435.579, Z    +0.000, E1  +334.614, E3 -423374.462}
SPL {X  -159.990, Y  +432.613, Z    +0.000, E1  +334.610, E3 -423387.729}
SPL {X  -159.990, Y  +429.079, Z    +0.000, E1  +334.593, E3 -423403.500}
SPL {X  -159.990, Y  +426.149, Z    +0.000, E1  +334.626, E3 -423416.662}
SPL {X  -159.990, Y  +423.417, Z    +0.000, E1  +334.600, E3 -423428.827}
SPL {X  -159.990, Y  +419.467, Z    +0.000, E1  +334.583, E3 -423446.462}
SPL {X  -159.990, Y  +415.368, Z    +0.000, E1  +334.593, E3 -423464.816}
SPL {X  -159.990, Y  +411.297, Z    +0.000, E1  +334.587, E3 -423483.012}
SPL {X  -159.990, Y  +407.450, Z    +0.000, E1  +334.599, E3 -423500.226}
SPL {X  -159.990, Y  +403.513, Z    +0.000, E1  +334.580, E3 -423517.780}
SPL {X  -159.990, Y  +399.294, Z    +0.000, E1  +334.582, E3 -423536.660}
SPL {X  -159.990, Y  +395.411, Z    +0.000, E1  +334.600, E3 -423554.074}
SPL {X  -159.990, Y  +392.473, Z    +0.000, E1  +334.623, E3 -423567.259}
SPL {X  -159.990, Y  +390.187, Z    +0.000, E1  +334.622, E3 -423577.517}
SPL {X  -159.990, Y  +387.503, Z    +0.000, E1  +334.622, E3 -423589.512}
SPL {X  -159.990, Y  +384.711, Z    +0.000, E1  +334.612, E3 -423601.956}
SPL {X  -159.988, Y  +381.794, Z    +0.000, E1  +334.611, E3 -423614.991}
SPL {X  -159.958, Y  +379.279, Z    +0.000, E1  +334.625, E3 -423626.281}
SPL {X  -159.894, Y  +376.959, Z    +0.000, E1  +334.630, E3 -423636.725}
SPL {X  -159.765, Y  +374.027, Z    +0.000, E1  +334.633, E3 -423649.941}
SPL {X  -159.607, Y  +371.442, Z    +0.000, E1  +334.673, E3 -423661.716}
SPL {X  -159.379, Y  +368.534, Z    +0.000, E1  +334.684, E3 -423674.904}
SPL {X  -159.113, Y  +365.767, Z    +0.000, E1  +334.734, E3 -423687.543}
SPL {X  -158.869, Y  +363.595, Z    +0.000, E1  +334.770, E3 -423697.514}
SPL {X  -158.527, Y  +360.915, Z    +0.000, E1  +334.798, E3 -423709.821}
SPL {X  -158.127, Y  +358.155, Z    +0.000, E1  +334.874, E3 -423722.659}
SPL {X  -158.095, Y  +357.947, Z    +0.000, E1  +338.259, E3 -423754.231}
ENDSPLINE

SPLINE
SPL {X  -158.454, Y  +360.384, Z    +0.000, E1  +340.634, E3 -423766.382}
SPL {X  -159.737, Y  +373.507, Z    +0.000, E1  +349.689, E3 -423788.417}
SPL {X  -159.990, Y  +382.574, Z    +0.000, E1  +355.537, E3 -423795.105}
SPL {X  -159.990, Y  +387.496, Z    +0.000, E1  +358.996, E3 -423797.850}
SPL {X  -159.990, Y  +395.121, Z    +0.000, E1  +364.514, E3 -423802.162}
SPL {X  -159.990, Y  +407.941, Z    +0.000, E1  +374.126, E3 -423814.237}
SPL {X  -159.990, Y  +418.671, Z    +0.000, E1  +379.855, E3 -423833.653}
SPL {X  -159.990, Y  +429.878, Z    +0.000, E1  +383.330, E3 -423863.708}
SPL {X  -159.990, Y  +432.103, Z    +0.000, E1  +383.301, E3 -423874.727}
SPL {X  -159.990, Y  +434.188, Z    +0.000, E1  +383.325, E3 -423884.923}
SPL {X  -159.990, Y  +436.320, Z    +0.000, E1  +383.304, E3 -423895.476}
SPL {X  -159.990, Y  +439.169, Z    +0.000, E1  +383.353, E3 -423909.393}
SPL {X  -159.990, Y  +442.945, Z    +0.000, E1  +383.339, E3 -423928.011}
SPL {X  -159.990, Y  +446.037, Z    +0.000, E1  +383.324, E3 -423943.261}
SPL {X  -159.990, Y  +448.341, Z    +0.000, E1  +383.317, E3 -423954.578}
SPL {X  -159.990, Y  +450.968, Z    +0.000, E1  +383.336, E3 -423967.494}
SPL {X  -159.990, Y  +454.421, Z    +0.000, E1  +383.348, E3 -423984.443}
SPL {X  -159.990, Y  +457.167, Z    +0.000, E1  +383.324, E3 -423997.986}
SPL {X  -159.990, Y  +459.480, Z    +0.000, E1  +383.323, E3 -424009.389}
SPL {X  -159.990, Y  +462.520, Z    +0.000, E1  +383.350, E3 -424024.294}
SPL {X  -159.990, Y  +465.602, Z    +0.000, E1  +383.328, E3 -424039.494}
SPL {X  -159.990, Y  +467.934, Z    +0.000, E1  +383.321, E3 -424050.988}
SPL {X  -159.990, Y  +469.939, Z    +0.000, E1  +383.319, E3 -424060.849}
SPL {X  -159.990, Y  +472.144, Z    +0.000, E1  +383.327, E3 -424071.700}
SPL {X  -159.990, Y  +474.152, Z    +0.000, E1  +383.309, E3 -424081.652}
SPL {X  -159.990, Y  +476.560, Z    +0.000, E1  +383.332, E3 -424093.460}
SPL {X  -159.990, Y  +478.770, Z    +0.000, E1  +383.306, E3 -424104.386}
SPL {X  -159.990, Y  +480.905, Z    +0.000, E1  +383.327, E3 -424114.854}
SPL {X  -159.990, Y  +484.251, Z    +0.000, E1  +383.352, E3 -424131.269}
SPL {X  -159.990, Y  +488.031, Z    +0.000, E1  +383.345, E3 -424149.902}
SPL {X  -159.990, Y  +491.121, Z    +0.000, E1  +383.323, E3 -424165.148}
SPL {X  -159.990, Y  +493.610, Z    +0.000, E1  +383.323, E3 -424177.401}
SPL {X  -159.990, Y  +496.863, Z    +0.000, E1  +383.350, E3 -424193.360}
SPL {X  -159.990, Y  +499.995, Z    +0.000, E1  +383.324, E3 -424208.822}
SPL {X  -159.990, Y  +502.341, Z    +0.000, E1  +383.320, E3 -424220.381}
SPL {X  -159.990, Y  +505.377, Z    +0.000, E1  +383.346, E3 -424235.271}
SPL {X  -159.990, Y  +508.024, Z    +0.000, E1  +383.315, E3 -424248.354}
SPL {X  -159.990, Y  +510.344, Z    +0.000, E1  +383.327, E3 -424259.761}
SPL {X  -159.990, Y  +513.289, Z    +0.000, E1  +383.332, E3 -424274.250}
SPL {X  -159.990, Y  +516.195, Z    +0.000, E1  +383.325, E3 -424288.569}
SPL {X  -159.990, Y  +518.925, Z    +0.000, E1  +383.333, E3 -424301.933}
SPL {X  -159.990, Y  +521.408, Z    +0.000, E1  +383.329, E3 -424314.142}
SPL {X  -159.990, Y  +523.942, Z    +0.000, E1  +383.333, E3 -424326.635}
SPL {X  -159.990, Y  +526.221, Z    +0.000, E1  +383.314, E3 -424337.911}
SPL {X  -159.990, Y  +527.834, Z    +0.000, E1  +383.311, E3 -424345.861}
SPL {X  -159.990, Y  +529.993, Z    +0.000, E1  +383.329, E3 -424356.437}
SPL {X  -159.990, Y  +532.441, Z    +0.000, E1  +383.322, E3 -424368.487}
SPL {X  -159.990, Y  +534.618, Z    +0.000, E1  +383.322, E3 -424379.220}
SPL {X  -159.990, Y  +537.024, Z    +0.000, E1  +383.321, E3 -424391.083}
SPL {X  -159.990, Y  +539.129, Z    +0.000, E1  +383.310, E3 -424401.466}
SPL {X  -159.990, Y  +541.183, Z    +0.000, E1  +383.319, E3 -424411.563}
SPL {X  -159.990, Y  +543.647, Z    +0.000, E1  +383.325, E3 -424423.665}
SPL {X  -159.990, Y  +546.832, Z    +0.000, E1  +383.349, E3 -424439.288}
SPL {X  -159.990, Y  +549.756, Z    +0.000, E1  +383.320, E3 -424453.729}
SPL {X  -159.990, Y  +551.655, Z    +0.000, E1  +383.320, E3 -424463.080}
SPL {X  -159.990, Y  +553.711, Z    +0.000, E1  +383.317, E3 -424473.202}
SPL {X  -159.990, Y  +555.637, Z    +0.000, E1  +383.323, E3 -424482.671}
SPL {X  -159.990, Y  +558.758, Z    +0.000, E1  +383.351, E3 -424497.980}
SPL {X  -159.990, Y  +561.830, Z    +0.000, E1  +383.325, E3 -424513.154}
SPL {X  -159.990, Y  +564.273, Z    +0.000, E1  +383.325, E3 -424525.178}
SPL {X  -159.990, Y  +567.351, Z    +0.000, E1  +383.348, E3 -424540.274}
SPL {X  -159.990, Y  +570.314, Z    +0.000, E1  +383.326, E3 -424554.906}
SPL {X  -159.990, Y  +572.504, Z    +0.000, E1  +383.321, E3 -424565.691}
SPL {X  -159.990, Y  +575.653, Z    +0.000, E1  +383.355, E3 -424581.128}
SPL {X  -159.990, Y  +578.932, Z    +0.000, E1  +383.330, E3 -424597.310}
SPL {X  -159.990, Y  +581.497, Z    +0.000, E1  +383.329, E3 -424609.895}
SPL {X  -159.990, Y  +583.973, Z    +0.000, E1  +383.332, E3 -424622.080}
SPL {X  -159.990, Y  +586.020, Z    +0.000, E1  +383.323, E3 -424632.164}
SPL {X  -159.990, Y  +587.711, Z    +0.000, E1  +383.318, E3 -424640.504}
SPL {X  -159.990, Y  +589.763, Z    +0.000, E1  +383.328, E3 -424650.580}
SPL {X  -159.990, Y  +591.698, Z    +0.000, E1  +383.324, E3 -424660.065}
SPL {X  -159.990, Y  +593.847, Z    +0.000, E1  +383.340, E3 -424670.595}
SPL {X  -159.990, Y  +597.018, Z    +0.000, E1  +383.367, E3 -424686.127}
SPL {X  -159.990, Y  +599.887, Z    +0.000, E1  +383.341, E3 -424700.231}
SPL {X  -159.990, Y  +601.949, Z    +0.000, E1  +383.344, E3 -424710.358}
SPL {X  -159.990, Y  +605.106, Z    +0.000, E1  +383.383, E3 -424725.804}
SPL {X  -159.990, Y  +608.111, Z    +0.000, E1  +383.342, E3 -424740.655}
SPL {X  -159.990, Y  +610.073, Z    +0.000, E1  +383.343, E3 -424750.313}
SPL {X  -159.990, Y  +612.330, Z    +0.000, E1  +383.340, E3 -424761.441}
SPL {X  -159.990, Y  +615.036, Z    +0.000, E1  +383.353, E3 -424774.728}
SPL {X  -159.990, Y  +618.481, Z    +0.000, E1  +383.366, E3 -424791.666}
SPL {X  -159.990, Y  +621.517, Z    +0.000, E1  +383.337, E3 -424806.649}
SPL {X  -159.990, Y  +623.764, Z    +0.000, E1  +383.335, E3 -424817.699}
SPL {X  -159.990, Y  +626.608, Z    +0.000, E1  +383.361, E3 -424831.624}
SPL {X  -159.990, Y  +630.271, Z    +0.000, E1  +383.375, E3 -424849.585}
SPL {X  -159.990, Y  +633.318, Z    +0.000, E1  +383.339, E3 -424864.663}
SPL {X  -159.990, Y  +635.650, Z    +0.000, E1  +383.339, E3 -424876.134}
SPL {X  -159.990, Y  +638.406, Z    +0.000, E1  +383.354, E3 -424889.700}
SPL {X  -159.990, Y  +641.831, Z    +0.000, E1  +383.342, E3 -424906.648}
SPL {X  -159.990, Y  +644.884, Z    +0.000, E1  +383.324, E3 -424921.735}
SPL {X  -159.990, Y  +647.550, Z    +0.000, E1  +383.318, E3 -424934.902}
SPL {X  -159.990, Y  +650.790, Z    +0.000, E1  +383.346, E3 -424950.768}
SPL {X  -159.990, Y  +654.543, Z    +0.000, E1  +383.348, E3 -424969.221}
SPL {X  -159.990, Y  +658.319, Z    +0.000, E1  +383.349, E3 -424987.811}
SPL {X  -159.990, Y  +661.392, Z    +0.000, E1  +383.318, E3 -425003.014}
SPL {X  -159.990, Y  +663.662, Z    +0.000, E1  +383.322, E3 -425014.138}
SPL {X  -159.990, Y  +665.964, Z    +0.000, E1  +383.328, E3 -425025.428}
SPL {X  -159.990, Y  +667.870, Z    +0.000, E1  +383.320, E3 -425034.835}
SPL {X  -159.990, Y  +669.861, Z    +0.000, E1  +383.321, E3 -425044.636}
SPL {X  -159.990, Y  +671.893, Z    +0.000, E1  +383.319, E3 -425054.644}
SPL {X  -159.974, Y  +673.789, Z    +0.000, E1  +383.323, E3 -425063.960}
SPL {X  -159.924, Y  +676.110, Z    +0.000, E1  +383.320, E3 -425075.445}
SPL {X  -159.801, Y  +679.265, Z    +0.000, E1  +383.327, E3 -425091.063}
SPL {X  -159.626, Y  +682.287, Z    +0.000, E1  +383.280, E3 -425106.162}
SPL {X  -159.462, Y  +684.486, Z    +0.000, E1  +383.258, E3 -425117.161}
SPL {X  -159.212, Y  +687.262, Z    +0.000, E1  +383.238, E3 -425131.065}
SPL {X  -158.971, Y  +689.529, Z    +0.000, E1  +383.181, E3 -425142.525}
SPL {X  -158.658, Y  +692.098, Z    +0.000, E1  +383.176, E3 -425155.432}
ENDSPLINE

SPLINE
SPL {X  -159.063, Y  +688.696, Z    +0.000, E1  +377.094, E3 -425197.650}
SPL {X  -159.957, Y  +674.769, Z    +0.000, E1  +367.092, E3 -425220.032}
SPL {X  -159.990, Y  +671.516, Z    +0.000, E1  +364.944, E3 -425222.418}
SPL {X  -159.990, Y  +663.928, Z    +0.000, E1  +359.662, E3 -425227.510}
SPL {X  -159.990, Y  +658.009, Z    +0.000, E1  +355.226, E3 -425231.209}
SPL {X  -159.990, Y  +651.879, Z    +0.000, E1  +350.548, E3 -425236.272}
SPL {X  -159.990, Y  +637.832, Z    +0.000, E1  +341.694, E3 -425253.863}
SPL {X  -159.990, Y  +626.634, Z    +0.000, E1  +337.968, E3 -425284.716}
SPL {X  -159.990, Y  +624.622, Z    +0.000, E1  +337.980, E3 -425295.300}
SPL {X  -159.990, Y  +622.489, Z    +0.000, E1  +337.969, E3 -425306.466}
SPL {X  -159.990, Y  +619.267, Z    +0.000, E1  +337.938, E3 -425323.300}
SPL {X  -159.990, Y  +615.467, Z    +0.000, E1  +337.940, E3 -425343.237}
SPL {X  -159.990, Y  +612.600, Z    +0.000, E1  +337.975, E3 -425358.347}
SPL {X  -159.990, Y  +610.646, Z    +0.000, E1  +337.979, E3 -425368.605}
SPL {X  -159.990, Y  +608.810, Z    +0.000, E1  +337.977, E3 -425378.238}
SPL {X  -159.990, Y  +605.804, Z    +0.000, E1  +337.936, E3 -425393.883}
SPL {X  -159.990, Y  +602.819, Z    +0.000, E1  +337.963, E3 -425409.554}
SPL {X  -159.990, Y  +600.642, Z    +0.000, E1  +337.968, E3 -425420.982}
SPL {X  -159.990, Y  +598.568, Z    +0.000, E1  +337.954, E3 -425431.775}
SPL {X  -159.990, Y  +596.440, Z    +0.000, E1  +337.964, E3 -425442.957}
SPL {X  -159.990, Y  +593.768, Z    +0.000, E1  +337.929, E3 -425456.889}
SPL {X  -159.990, Y  +590.068, Z    +0.000, E1  +337.924, E3 -425476.258}
SPL {X  -159.990, Y  +586.620, Z    +0.000, E1  +337.935, E3 -425494.320}
SPL {X  -159.990, Y  +584.080, Z    +0.000, E1  +337.953, E3 -425507.647}
SPL {X  -159.990, Y  +581.924, Z    +0.000, E1  +337.949, E3 -425518.947}
SPL {X  -159.990, Y  +578.886, Z    +0.000, E1  +337.918, E3 -425534.801}
SPL {X  -159.990, Y  +576.252, Z    +0.000, E1  +337.962, E3 -425548.699}
SPL {X  -159.990, Y  +574.188, Z    +0.000, E1  +337.947, E3 -425559.472}
SPL {X  -159.990, Y  +571.954, Z    +0.000, E1  +337.959, E3 -425571.229}
SPL {X  -159.990, Y  +570.110, Z    +0.000, E1  +337.958, E3 -425580.880}
SPL {X  -159.990, Y  +568.165, Z    +0.000, E1  +337.957, E3 -425591.060}
SPL {X  -159.990, Y  +565.292, Z    +0.000, E1  +337.922, E3 -425606.038}
SPL {X  -159.990, Y  +562.598, Z    +0.000, E1  +337.958, E3 -425620.249}
SPL {X  -159.990, Y  +560.652, Z    +0.000, E1  +337.962, E3 -425630.461}
SPL {X  -159.990, Y  +558.143, Z    +0.000, E1  +337.928, E3 -425643.493}
SPL {X  -159.990, Y  +555.329, Z    +0.000, E1  +337.943, E3 -425658.237}
SPL {X  -159.990, Y  +553.115, Z    +0.000, E1  +337.946, E3 -425669.842}
SPL {X  -159.990, Y  +550.886, Z    +0.000, E1  +337.944, E3 -425681.524}
SPL {X  -159.990, Y  +548.568, Z    +0.000, E1  +337.944, E3 -425693.645}
SPL {X  -159.990, Y  +546.537, Z    +0.000, E1  +337.948, E3 -425704.280}
SPL {X  -159.990, Y  +545.062, Z    +0.000, E1  +337.955, E3 -425712.038}
SPL {X  -159.990, Y  +543.060, Z    +0.000, E1  +337.943, E3 -425722.518}
SPL {X  -159.990, Y  +539.928, Z    +0.000, E1  +337.917, E3 -425738.859}
SPL {X  -159.990, Y  +536.935, Z    +0.000, E1  +337.942, E3 -425754.576}
SPL {X  -159.990, Y  +534.656, Z    +0.000, E1  +337.946, E3 -425766.519}
SPL {X  -159.990, Y  +532.453, Z    +0.000, E1  +337.944, E3 -425778.047}
SPL {X  -159.990, Y  +530.660, Z    +0.000, E1  +337.952, E3 -425787.449}
SPL {X  -159.990, Y  +528.702, Z    +0.000, E1  +337.939, E3 -425797.662}
SPL {X  -159.990, Y  +525.760, Z    +0.000, E1  +337.914, E3 -425813.004}
SPL {X  -159.990, Y  +522.838, Z    +0.000, E1  +337.933, E3 -425828.370}
SPL {X  -159.990, Y  +519.698, Z    +0.000, E1  +337.916, E3 -425844.753}
SPL {X  -159.990, Y  +517.251, Z    +0.000, E1  +337.946, E3 -425857.613}
SPL {X  -159.990, Y  +515.568, Z    +0.000, E1  +338.084, E3 -425867.710}
ENDSPLINE

SPLINE
SPL {X  -159.990, Y  +517.293, Z    +0.000, E1  +340.923, E3 -425884.008}
ENDSPLINE

SPLINE
SPL {X  -159.990, Y  +512.548, Z    +0.000, E1  +339.587, E3 -425899.583}
SPL {X  -159.990, Y  +508.660, Z    +0.000, E1  +338.515, E3 -425911.638}
SPL {X  -159.990, Y  +503.499, Z    +0.000, E1  +337.116, E3 -425926.717}
SPL {X  -159.990, Y  +498.406, Z    +0.000, E1  +335.789, E3 -425940.750}
SPL {X  -159.990, Y  +494.693, Z    +0.000, E1  +334.929, E3 -425951.217}
SPL {X  -159.990, Y  +491.649, Z    +0.000, E1  +334.596, E3 -425962.420}
SPL {X  -159.990, Y  +488.807, Z    +0.000, E1  +334.603, E3 -425975.144}
SPL {X  -159.990, Y  +486.070, Z    +0.000, E1  +334.601, E3 -425987.375}
SPL {X  -159.990, Y  +483.747, Z    +0.000, E1  +334.616, E3 -425997.788}
SPL {X  -159.990, Y  +481.038, Z    +0.000, E1  +334.588, E3 -426009.844}
SPL {X  -159.990, Y  +478.407, Z    +0.000, E1  +334.616, E3 -426021.657}
SPL {X  -159.990, Y  +475.940, Z    +0.000, E1  +334.597, E3 -426032.648}
SPL {X  -159.990, Y  +473.026, Z    +0.000, E1  +334.601, E3 -426045.677}
SPL {X  -159.990, Y  +470.047, Z    +0.000, E1  +334.598, E3 -426058.996}
SPL {X  -159.990, Y  +467.082, Z    +0.000, E1  +334.601, E3 -426072.243}
SPL {X  -159.990, Y  +464.919, Z    +0.000, E1  +334.619, E3 -426081.970}
SPL {X  -159.990, Y  +462.520, Z    +0.000, E1  +334.600, E3 -426092.644}
SPL {X  -159.990, Y  +460.081, Z    +0.000, E1  +334.610, E3 -426103.546}
SPL {X  -159.990, Y  +457.497, Z    +0.000, E1  +334.597, E3 -426115.070}
SPL {X  -159.990, Y  +454.323, Z    +0.000, E1  +334.588, E3 -426129.229}
SPL {X  -159.990, Y  +451.400, Z    +0.000, E1  +334.603, E3 -426142.320}
SPL {X  -159.990, Y  +448.503, Z    +0.000, E1  +334.590, E3 -426155.238}
SPL {X  -159.990, Y  +445.882, Z    +0.000, E1  +334.615, E3 -426167.040}
SPL {X  -159.990, Y  +443.345, Z    +0.000, E1  +334.610, E3 -426178.422}
SPL {X  -159.990, Y  +441.077, Z    +0.000, E1  +334.631, E3 -426188.621}
SPL {X  -159.990, Y  +438.608, Z    +0.000, E1  +334.608, E3 -426199.617}
SPL {X  -159.990, Y  +434.852, Z    +0.000, E1  +334.585, E3 -426216.372}
SPL {X  -159.990, Y  +430.645, Z    +0.000, E1  +334.586, E3 -426235.191}
SPL {X  -159.990, Y  +426.865, Z    +0.000, E1  +334.602, E3 -426252.121}
SPL {X  -159.990, Y  +423.417, Z    +0.000, E1  +334.600, E3 -426267.537}
SPL {X  -159.990, Y  +419.467, Z    +0.000, E1  +334.583, E3 -426285.172}
SPL {X  -159.990, Y  +416.355, Z    +0.000, E1  +334.625, E3 -426299.169}
SPL {X  -159.990, Y  +413.684, Z    +0.000, E1  +334.603, E3 -426311.076}
SPL {X  -159.990, Y  +410.645, Z    +0.000, E1  +334.615, E3 -426324.687}
SPL {X  -159.990, Y  +408.351, Z    +0.000, E1  +334.628, E3 -426334.974}
SPL {X  -159.990, Y  +406.574, Z    +0.000, E1  +334.625, E3 -426342.890}
SPL {X  -159.990, Y  +404.255, Z    +0.000, E1  +334.609, E3 -426353.227}
SPL {X  -159.990, Y  +401.103, Z    +0.000, E1  +334.596, E3 -426367.291}
SPL {X  -159.990, Y  +398.389, Z    +0.000, E1  +334.619, E3 -426379.487}
SPL {X  -159.990, Y  +395.411, Z    +0.000, E1  +334.600, E3 -426392.784}
SPL {X  -159.990, Y  +392.473, Z    +0.000, E1  +334.623, E3 -426405.969}
SPL {X  -159.990, Y  +390.187, Z    +0.000, E1  +334.622, E3 -426416.227}
SPL {X  -159.990, Y  +387.503, Z    +0.000, E1  +334.622, E3 -426428.222}
SPL {X  -159.990, Y  +384.711, Z    +0.000, E1  +334.612, E3 -426440.666}
SPL {X  -159.988, Y  +381.794, Z    +0.000, E1  +334.611, E3 -426453.700}
SPL {X  -159.958, Y  +379.279, Z    +0.000, E1  +334.625, E3 -426464.991}
SPL {X  -159.867, Y  +376.223, Z    +0.000, E1  +334.608, E3 -426478.705}
SPL {X  -159.727, Y  +373.325, Z    +0.000, E1  +334.659, E3 -426491.870}
SPL {X  -159.549, Y  +370.634, Z    +0.000, E1  +334.653, E3 -426504.043}
SPL {X  -159.201, Y  +366.633, Z    +0.000, E1  +334.686, E3 -426522.235}
SPL {X  -158.798, Y  +363.007, Z    +0.000, E1  +334.761, E3 -426538.893}
SPL {X  -158.453, Y  +360.380, Z    +0.000, E1  +334.828, E3 -426551.038}
SPL {X  -158.127, Y  +358.155, Z    +0.000, E1  +334.874, E3 -426561.368}
SPL {X  -158.095, Y  +357.947, Z    +0.000, E1  +338.259, E3 -426592.941}
ENDSPLINE

SPLINE
SPL {X  -158.454, Y  +360.384, Z    +0.000, E1  +340.634, E3 -426605.092}
SPL {X  -159.737, Y  +373.507, Z    +0.000, E1  +349.689, E3 -426627.127}
SPL {X  -159.990, Y  +382.574, Z    +0.000, E1  +355.537, E3 -426633.815}
SPL {X  -159.990, Y  +389.909, Z    +0.000, E1  +360.662, E3 -426637.829}
SPL {X  -159.990, Y  +396.289, Z    +0.000, E1  +365.500, E3 -426641.610}
SPL {X  -159.990, Y  +407.941, Z    +0.000, E1  +374.126, E3 -426652.946}
SPL {X  -159.990, Y  +418.671, Z    +0.000, E1  +379.855, E3 -426672.363}
SPL {X  -159.990, Y  +429.878, Z    +0.000, E1  +383.330, E3 -426702.418}
SPL {X  -159.990, Y  +432.103, Z    +0.000, E1  +383.301, E3 -426713.436}
SPL {X  -159.990, Y  +434.188, Z    +0.000, E1  +383.325, E3 -426723.633}
SPL {X  -159.990, Y  +436.320, Z    +0.000, E1  +383.304, E3 -426734.186}
SPL {X  -159.990, Y  +439.169, Z    +0.000, E1  +383.353, E3 -426748.103}
SPL {X  -159.990, Y  +442.945, Z    +0.000, E1  +383.339, E3 -426766.720}
SPL {X  -159.990, Y  +446.037, Z    +0.000, E1  +383.324, E3 -426781.971}
SPL {X  -159.990, Y  +448.341, Z    +0.000, E1  +383.317, E3 -426793.288}
SPL {X  -159.990, Y  +450.345, Z    +0.000, E1  +383.316, E3 -426803.166}
SPL {X  -159.990, Y  +452.828, Z    +0.000, E1  +383.330, E3 -426815.366}
SPL {X  -159.990, Y  +456.338, Z    +0.000, E1  +383.359, E3 -426832.558}
SPL {X  -159.990, Y  +459.480, Z    +0.000, E1  +383.323, E3 -426848.099}
SPL {X  -159.990, Y  +461.803, Z    +0.000, E1  +383.322, E3 -426859.534}
SPL {X  -159.990, Y  +464.971, Z    +0.000, E1  +383.357, E3 -426875.040}
SPL {X  -159.990, Y  +467.934, Z    +0.000, E1  +383.321, E3 -426889.698}
SPL {X  -159.990, Y  +469.939, Z    +0.000, E1  +383.319, E3 -426899.559}
SPL {X  -159.990, Y  +472.144, Z    +0.000, E1  +383.327, E3 -426910.410}
SPL {X  -159.990, Y  +474.994, Z    +0.000, E1  +383.334, E3 -426924.458}
SPL {X  -159.990, Y  +477.323, Z    +0.000, E1  +383.307, E3 -426935.973}
SPL {X  -159.990, Y  +479.553, Z    +0.000, E1  +383.328, E3 -426946.909}
SPL {X  -159.990, Y  +482.799, Z    +0.000, E1  +383.343, E3 -426962.848}
SPL {X  -159.990, Y  +485.299, Z    +0.000, E1  +383.310, E3 -426975.233}
SPL {X  -159.990, Y  +488.031, Z    +0.000, E1  +383.345, E3 -426988.612}
SPL {X  -159.990, Y  +491.121, Z    +0.000, E1  +383.323, E3 -427003.857}
SPL {X  -159.990, Y  +493.610, Z    +0.000, E1  +383.323, E3 -427016.110}
SPL {X  -159.990, Y  +496.863, Z    +0.000, E1  +383.350, E3 -427032.070}
SPL {X  -159.990, Y  +499.995, Z    +0.000, E1  +383.324, E3 -427047.532}
SPL {X  -159.990, Y  +502.341, Z    +0.000, E1  +383.320, E3 -427059.091}
SPL {X  -159.990, Y  +505.377, Z    +0.000, E1  +383.346, E3 -427073.981}
SPL {X  -159.990, Y  +508.697, Z    +0.000, E1  +383.335, E3 -427090.341}
SPL {X  -159.990, Y  +511.771, Z    +0.000, E1  +383.331, E3 -427105.488}
SPL {X  -159.990, Y  +514.016, Z    +0.000, E1  +383.308, E3 -427116.591}
SPL {X  -159.990, Y  +516.195, Z    +0.000, E1  +383.325, E3 -427127.279}
SPL {X  -159.990, Y  +518.925, Z    +0.000, E1  +383.333, E3 -427140.643}
SPL {X  -159.990, Y  +521.408, Z    +0.000, E1  +383.329, E3 -427152.852}
SPL {X  -159.990, Y  +523.942, Z    +0.000, E1  +383.333, E3 -427165.344}
SPL {X  -159.990, Y  +526.221, Z    +0.000, E1  +383.314, E3 -427176.620}
SPL {X  -159.990, Y  +527.834, Z    +0.000, E1  +383.311, E3 -427184.570}
SPL {X  -159.990, Y  +529.993, Z    +0.000, E1  +383.329, E3 -427195.146}
SPL {X  -159.990, Y  +532.441, Z    +0.000, E1  +383.322, E3 -427207.197}
SPL {X  -159.990, Y  +534.618, Z    +0.000, E1  +383.322, E3 -427217.930}
SPL {X  -159.990, Y  +537.024, Z    +0.000, E1  +383.321, E3 -427229.792}
SPL {X  -159.990, Y  +539.129, Z    +0.000, E1  +383.310, E3 -427240.175}
SPL {X  -159.990, Y  +541.183, Z    +0.000, E1  +383.319, E3 -427250.272}
SPL {X  -159.990, Y  +543.647, Z    +0.000, E1  +383.325, E3 -427262.375}
SPL {X  -159.990, Y  +546.832, Z    +0.000, E1  +383.349, E3 -427277.998}
SPL {X  -159.990, Y  +549.756, Z    +0.000, E1  +383.320, E3 -427292.439}
SPL {X  -159.990, Y  +551.655, Z    +0.000, E1  +383.320, E3 -427301.790}
SPL {X  -159.990, Y  +553.711, Z    +0.000, E1  +383.317, E3 -427311.912}
SPL {X  -159.990, Y  +555.637, Z    +0.000, E1  +383.323, E3 -427321.380}
SPL {X  -159.990, Y  +558.758, Z    +0.000, E1  +383.351, E3 -427336.690}
SPL {X  -159.990, Y  +561.830, Z    +0.000, E1  +383.325, E3 -427351.863}
SPL {X  -159.990, Y  +564.273, Z    +0.000, E1  +383.325, E3 -427363.888}
SPL {X  -159.990, Y  +567.351, Z    +0.000, E1  +383.348, E3 -427378.983}
SPL {X  -159.990, Y  +570.314, Z    +0.000, E1  +383.326, E3 -427393.615}
SPL {X  -159.990, Y  +572.504, Z    +0.000, E1  +383.321, E3 -427404.400}
SPL {X  -159.990, Y  +575.653, Z    +0.000, E1  +383.355, E3 -427419.837}
SPL {X  -159.990, Y  +578.932, Z    +0.000, E1  +383.330, E3 -427436.020}
SPL {X  -159.990, Y  +581.497, Z    +0.000, E1  +383.329, E3 -427448.605}
SPL {X  -159.990, Y  +583.973, Z    +0.000, E1  +383.332, E3 -427460.790}
SPL {X  -159.990, Y  +586.877, Z    +0.000, E1  +383.349, E3 -427475.044}
SPL {X  -159.990, Y  +590.594, Z    +0.000, E1  +383.363, E3 -427493.295}
SPL {X  -159.990, Y  +593.847, Z    +0.000, E1  +383.340, E3 -427509.305}
SPL {X  -159.990, Y  +596.027, Z    +0.000, E1  +383.330, E3 -427520.051}
SPL {X  -159.990, Y  +599.017, Z    +0.000, E1  +383.373, E3 -427534.616}
SPL {X  -159.990, Y  +601.949, Z    +0.000, E1  +383.344, E3 -427549.068}
SPL {X  -159.990, Y  +604.315, Z    +0.000, E1  +383.350, E3 -427560.693}
SPL {X  -159.990, Y  +607.388, Z    +0.000, E1  +383.369, E3 -427575.758}
SPL {X  -159.990, Y  +610.073, Z    +0.000, E1  +383.343, E3 -427589.023}
SPL {X  -159.990, Y  +613.021, Z    +0.000, E1  +383.365, E3 -427603.494}
SPL {X  -159.990, Y  +615.657, Z    +0.000, E1  +383.331, E3 -427616.542}
SPL {X  -159.990, Y  +617.658, Z    +0.000, E1  +383.335, E3 -427626.384}
SPL {X  -159.990, Y  +620.788, Z    +0.000, E1  +383.368, E3 -427641.717}
SPL {X  -159.990, Y  +624.347, Z    +0.000, E1  +383.355, E3 -427659.237}
SPL {X  -159.990, Y  +627.144, Z    +0.000, E1  +383.340, E3 -427673.007}
SPL {X  -159.990, Y  +629.284, Z    +0.000, E1  +383.339, E3 -427683.515}
SPL {X  -159.990, Y  +631.206, Z    +0.000, E1  +383.337, E3 -427692.968}
SPL {X  -159.990, Y  +633.318, Z    +0.000, E1  +383.339, E3 -427703.373}
SPL {X  -159.990, Y  +635.650, Z    +0.000, E1  +383.339, E3 -427714.843}
SPL {X  -159.990, Y  +637.597, Z    +0.000, E1  +383.330, E3 -427724.466}
SPL {X  -159.990, Y  +640.369, Z    +0.000, E1  +383.354, E3 -427738.100}
SPL {X  -159.990, Y  +644.241, Z    +0.000, E1  +383.355, E3 -427757.212}
SPL {X  -159.990, Y  +648.287, Z    +0.000, E1  +383.349, E3 -427777.169}
SPL {X  -159.990, Y  +651.427, Z    +0.000, E1  +383.319, E3 -427792.664}
SPL {X  -159.990, Y  +653.536, Z    +0.000, E1  +383.313, E3 -427803.046}
SPL {X  -159.990, Y  +656.380, Z    +0.000, E1  +383.347, E3 -427816.982}
SPL {X  -159.990, Y  +659.180, Z    +0.000, E1  +383.314, E3 -427830.830}
SPL {X  -159.990, Y  +661.392, Z    +0.000, E1  +383.318, E3 -427841.723}
SPL {X  -159.990, Y  +663.662, Z    +0.000, E1  +383.322, E3 -427852.848}
SPL {X  -159.990, Y  +665.964, Z    +0.000, E1  +383.328, E3 -427864.138}
SPL {X  -159.990, Y  +668.989, Z    +0.000, E1  +383.359, E3 -427878.974}
SPL {X  -159.983, Y  +672.946, Z    +0.000, E1  +383.359, E3 -427898.455}
SPL {X  -159.924, Y  +676.110, Z    +0.000, E1  +383.320, E3 -427914.154}
SPL {X  -159.845, Y  +678.302, Z    +0.000, E1  +383.298, E3 -427925.056}
SPL {X  -159.760, Y  +680.081, Z    +0.000, E1  +383.288, E3 -427933.900}
SPL {X  -159.626, Y  +682.287, Z    +0.000, E1  +383.280, E3 -427944.871}
SPL {X  -159.462, Y  +684.486, Z    +0.000, E1  +383.258, E3 -427955.871}
SPL {X  -159.212, Y  +687.262, Z    +0.000, E1  +383.238, E3 -427969.775}
SPL {X  -158.861, Y  +690.475, Z    +0.000, E1  +383.199, E3 -427985.943}
SPL {X  -158.553, Y  +692.896, Z    +0.000, E1  +383.130, E3 -427998.239}
ENDSPLINE

SPLINE
SPL {X  -159.063, Y  +688.696, Z    +0.000, E1  +377.094, E3 -428036.360}
SPL {X  -159.987, Y  +672.488, Z    +0.000, E1  +365.638, E3 -428060.425}
SPL {X  -159.990, Y  +663.928, Z    +0.000, E1  +359.662, E3 -428066.219}
SPL {X  -159.990, Y  +658.009, Z    +0.000, E1  +355.226, E3 -428069.919}
SPL {X  -159.990, Y  +651.879, Z    +0.000, E1  +350.548, E3 -428074.982}
SPL {X  -159.990, Y  +637.832, Z    +0.000, E1  +341.694, E3 -428092.573}
SPL {X  -159.990, Y  +626.634, Z    +0.000, E1  +337.968, E3 -428123.426}
SPL {X  -159.990, Y  +624.622, Z    +0.000, E1  +337.980, E3 -428134.010}
SPL {X  -159.990, Y  +622.489, Z    +0.000, E1  +337.969, E3 -428145.176}
SPL {X  -159.990, Y  +619.955, Z    +0.000, E1  +337.968, E3 -428158.466}
SPL {X  -159.990, Y  +617.386, Z    +0.000, E1  +337.968, E3 -428171.941}
SPL {X  -159.990, Y  +614.863, Z    +0.000, E1  +337.969, E3 -428185.173}
SPL {X  -159.990, Y  +612.600, Z    +0.000, E1  +337.975, E3 -428197.057}
SPL {X  -159.990, Y  +610.646, Z    +0.000, E1  +337.979, E3 -428207.314}
SPL {X  -159.990, Y  +608.810, Z    +0.000, E1  +337.977, E3 -428216.947}
SPL {X  -159.990, Y  +605.804, Z    +0.000, E1  +337.936, E3 -428232.593}
SPL {X  -159.990, Y  +602.819, Z    +0.000, E1  +337.963, E3 -428248.264}
SPL {X  -159.990, Y  +600.642, Z    +0.000, E1  +337.968, E3 -428259.692}
SPL {X  -159.990, Y  +598.568, Z    +0.000, E1  +337.954, E3 -428270.485}
SPL {X  -159.990, Y  +596.440, Z    +0.000, E1  +337.964, E3 -428281.666}
SPL {X  -159.990, Y  +593.768, Z    +0.000, E1  +337.929, E3 -428295.599}
SPL {X  -159.990, Y  +590.068, Z    +0.000, E1  +337.924, E3 -428314.967}
SPL {X  -159.990, Y  +586.620, Z    +0.000, E1  +337.935, E3 -428333.030}
SPL {X  -159.990, Y  +584.080, Z    +0.000, E1  +337.953, E3 -428346.356}
SPL {X  -159.990, Y  +581.924, Z    +0.000, E1  +337.949, E3 -428357.657}
SPL {X  -159.990, Y  +578.886, Z    +0.000, E1  +337.918, E3 -428373.511}
SPL {X  -159.990, Y  +576.252, Z    +0.000, E1  +337.962, E3 -428387.409}
SPL {X  -159.990, Y  +574.188, Z    +0.000, E1  +337.947, E3 -428398.182}
SPL {X  -159.990, Y  +571.954, Z    +0.000, E1  +337.959, E3 -428409.939}
SPL {X  -159.990, Y  +570.110, Z    +0.000, E1  +337.958, E3 -428419.590}
SPL {X  -159.990, Y  +568.165, Z    +0.000, E1  +337.957, E3 -428429.769}
SPL {X  -159.990, Y  +565.292, Z    +0.000, E1  +337.922, E3 -428444.747}
SPL {X  -159.990, Y  +562.598, Z    +0.000, E1  +337.958, E3 -428458.959}
SPL {X  -159.990, Y  +560.652, Z    +0.000, E1  +337.962, E3 -428469.171}
SPL {X  -159.990, Y  +558.143, Z    +0.000, E1  +337.928, E3 -428482.202}
SPL {X  -159.990, Y  +555.329, Z    +0.000, E1  +337.943, E3 -428496.947}
SPL {X  -159.990, Y  +553.115, Z    +0.000, E1  +337.946, E3 -428508.552}
SPL {X  -159.990, Y  +550.886, Z    +0.000, E1  +337.944, E3 -428520.233}
SPL {X  -159.990, Y  +548.568, Z    +0.000, E1  +337.944, E3 -428532.354}
SPL {X  -159.990, Y  +546.537, Z    +0.000, E1  +337.948, E3 -428542.989}
SPL {X  -159.990, Y  +545.062, Z    +0.000, E1  +337.955, E3 -428550.748}
SPL {X  -159.990, Y  +543.060, Z    +0.000, E1  +337.943, E3 -428561.227}
SPL {X  -159.990, Y  +539.928, Z    +0.000, E1  +337.917, E3 -428577.569}
SPL {X  -159.990, Y  +536.935, Z    +0.000, E1  +337.942, E3 -428593.286}
SPL {X  -159.990, Y  +534.656, Z    +0.000, E1  +337.946, E3 -428605.229}
SPL {X  -159.990, Y  +531.679, Z    +0.000, E1  +337.913, E3 -428620.743}
SPL {X  -159.990, Y  +527.941, Z    +0.000, E1  +337.907, E3 -428640.285}
SPL {X  -159.990, Y  +524.425, Z    +0.000, E1  +337.922, E3 -428658.741}
SPL {X  -159.990, Y  +521.385, Z    +0.000, E1  +337.932, E3 -428674.684}
SPL {X  -159.990, Y  +518.216, Z    +0.000, E1  +337.909, E3 -428691.190}
SPL {X  -159.990, Y  +515.568, Z    +0.000, E1  +338.084, E3 -428706.420}
ENDSPLINE

SPLINE
SPL {X  -159.990, Y  +518.374, Z    +0.000, E1  +341.240, E3 -428719.008}
ENDSPLINE

SPLINE
SPL {X  -159.990, Y  +513.606, Z    +0.000, E1  +339.879, E3 -428734.918}
SPL {X  -159.990, Y  +508.660, Z    +0.000, E1  +338.515, E3 -428750.348}
SPL {X  -159.990, Y  +505.237, Z    +0.000, E1  +337.606, E3 -428760.605}
SPL {X  -159.990, Y  +501.963, Z    +0.000, E1  +336.712, E3 -428769.709}
SPL {X  -159.990, Y  +498.406, Z    +0.000, E1  +335.789, E3 -428779.460}
SPL {X  -159.990, Y  +494.693, Z    +0.000, E1  +334.929, E3 -428789.927}
SPL {X  -159.990, Y  +491.649, Z    +0.000, E1  +334.596, E3 -428801.130}
SPL {X  -159.990, Y  +488.807, Z    +0.000, E1  +334.603, E3 -428813.854}
SPL {X  -159.990, Y  +486.070, Z    +0.000, E1  +334.601, E3 -428826.085}
SPL {X  -159.990, Y  +482.821, Z    +0.000, E1  +334.589, E3 -428840.586}
SPL {X  -159.990, Y  +480.183, Z    +0.000, E1  +334.616, E3 -428852.427}
SPL {X  -159.990, Y  +477.508, Z    +0.000, E1  +334.590, E3 -428864.335}
SPL {X  -159.990, Y  +473.634, Z    +0.000, E1  +334.574, E3 -428881.625}
SPL {X  -159.990, Y  +470.047, Z    +0.000, E1  +334.598, E3 -428897.705}
SPL {X  -159.990, Y  +466.213, Z    +0.000, E1  +334.567, E3 -428914.785}
SPL {X  -159.990, Y  +462.520, Z    +0.000, E1  +334.600, E3 -428931.354}
SPL {X  -159.990, Y  +460.081, Z    +0.000, E1  +334.610, E3 -428942.255}
SPL {X  -159.990, Y  +457.497, Z    +0.000, E1  +334.597, E3 -428953.780}
SPL {X  -159.990, Y  +455.126, Z    +0.000, E1  +334.611, E3 -428964.388}
SPL {X  -159.990, Y  +452.123, Z    +0.000, E1  +334.574, E3 -428977.746}
SPL {X  -159.990, Y  +448.503, Z    +0.000, E1  +334.590, E3 -428993.947}
SPL {X  -159.990, Y  +445.882, Z    +0.000, E1  +334.615, E3 -429005.750}
SPL {X  -159.990, Y  +443.345, Z    +0.000, E1  +334.610, E3 -429017.132}
SPL {X  -159.990, Y  +441.077, Z    +0.000, E1  +334.631, E3 -429027.330}
SPL {X  -159.990, Y  +438.608, Z    +0.000, E1  +334.608, E3 -429038.327}
SPL {X  -159.990, Y  +435.579, Z    +0.000, E1  +334.614, E3 -429051.881}
SPL {X  -159.990, Y  +432.613, Z    +0.000, E1  +334.610, E3 -429065.149}
SPL {X  -159.990, Y  +429.079, Z    +0.000, E1  +334.593, E3 -429080.919}
SPL {X  -159.990, Y  +426.149, Z    +0.000, E1  +334.626, E3 -429094.081}
SPL {X  -159.990, Y  +423.417, Z    +0.000, E1  +334.600, E3 -429106.247}
SPL {X  -159.990, Y  +419.467, Z    +0.000, E1  +334.583, E3 -429123.882}
SPL {X  -159.990, Y  +415.368, Z    +0.000, E1  +334.593, E3 -429142.236}
SPL {X  -159.990, Y  +411.297, Z    +0.000, E1  +334.587, E3 -429160.431}
SPL {X  -159.990, Y  +407.450, Z    +0.000, E1  +334.599, E3 -429177.646}
SPL {X  -159.990, Y  +403.513, Z    +0.000, E1  +334.580, E3 -429195.199}
SPL {X  -159.990, Y  +400.403, Z    +0.000, E1  +334.620, E3 -429209.182}
SPL {X  -159.990, Y  +397.743, Z    +0.000, E1  +334.600, E3 -429221.051}
SPL {X  -159.990, Y  +394.848, Z    +0.000, E1  +334.621, E3 -429234.052}
SPL {X  -159.990, Y  +392.473, Z    +0.000, E1  +334.623, E3 -429244.679}
SPL {X  -159.990, Y  +390.187, Z    +0.000, E1  +334.622, E3 -429254.937}
SPL {X  -159.990, Y  +387.503, Z    +0.000, E1  +334.622, E3 -429266.932}
SPL {X  -159.990, Y  +384.711, Z    +0.000, E1  +334.612, E3 -429279.375}
SPL {X  -159.988, Y  +381.794, Z    +0.000, E1  +334.611, E3 -429292.410}
SPL {X  -159.958, Y  +379.279, Z    +0.000, E1  +334.625, E3 -429303.700}
SPL {X  -159.894, Y  +376.959, Z    +0.000, E1  +334.630, E3 -429314.145}
SPL {X  -159.765, Y  +374.027, Z    +0.000, E1  +334.633, E3 -429327.360}
SPL {X  -159.607, Y  +371.442, Z    +0.000, E1  +334.673, E3 -429339.135}
SPL {X  -159.379, Y  +368.534, Z    +0.000, E1  +334.684, E3 -429352.323}
SPL {X  -159.113, Y  +365.767, Z    +0.000, E1  +334.734, E3 -429364.962}
SPL {X  -158.798, Y  +363.007, Z    +0.000, E1  +334.761, E3 -429377.603}
SPL {X  -158.453, Y  +360.380, Z    +0.000, E1  +334.828, E3 -429389.747}
SPL {X  -158.127, Y  +358.155, Z    +0.000, E1  +334.874, E3 -429400.078}
SPL {X  -158.095, Y  +357.947, Z    +0.000, E1  +338.259, E3 -429431.650}
ENDSPLINE

